Yaskawa INFORM job: A_ROOF_SIDE_0617_2_PAINT_56.JBI

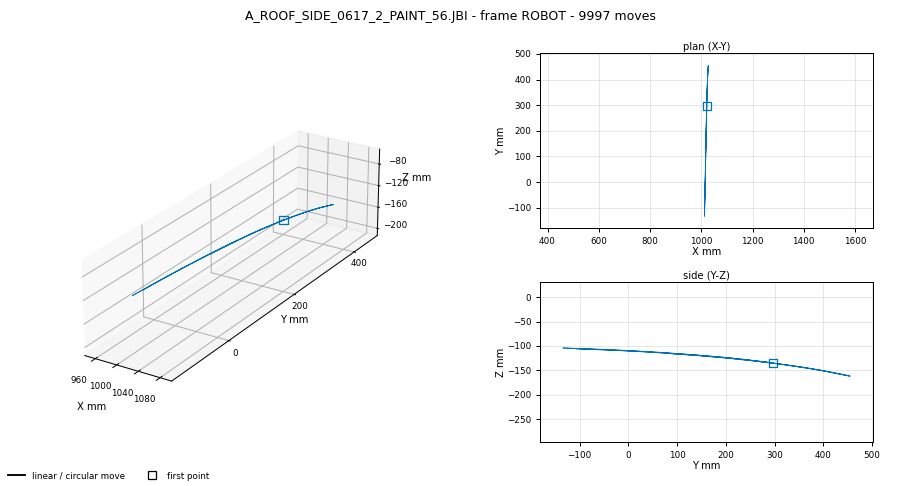
[picture p0: tool path of A_ROOF_SIDE_0617_2_PAINT_56.JBI in frame ROBOT, 9997 of 9997 moves have a stored position in this frame; points joined in program order, loops and branches not executed]
/JOB
//NAME A_ROOF_SIDE_0617_2_PAINT56
//POS
///NPOS 9997,0,0,0,0,0
///TOOL 1
///USER 0
///POSTYPE ROBOT
///RECTAN
///RCONF 1,0,0,0,0,0,0,0,0,0,0,0,0,0,0,0,0,0,0,0,0,0,0,0
C00000=1021.853,296.676,-134.515,170.306,49.131,159.506
C00001=1021.846,296.428,-134.484,170.301,49.134,159.506
C00002=1021.840,296.180,-134.452,170.296,49.136,159.506
C00003=1021.834,295.932,-134.419,170.291,49.139,159.506
C00004=1021.827,295.684,-134.388,170.287,49.142,159.506
C00005=1021.821,295.436,-134.355,170.281,49.145,159.506
C00006=1021.814,295.189,-134.324,170.276,49.148,159.506
C00007=1021.808,294.940,-134.292,170.271,49.151,159.506
C00008=1021.802,294.693,-134.259,170.266,49.153,159.505
C00009=1021.795,294.445,-134.227,170.261,49.156,159.505
C00010=1021.789,294.197,-134.195,170.256,49.159,159.505
C00011=1021.782,293.949,-134.163,170.251,49.162,159.505
C00012=1021.776,293.701,-134.131,170.246,49.165,159.505
C00013=1021.770,293.476,-134.103,170.242,49.168,159.505
C00014=1021.765,293.252,-134.073,170.237,49.170,159.505
C00015=1021.758,293.027,-134.045,170.233,49.173,159.505
C00016=1021.753,292.802,-134.016,170.227,49.176,159.505
C00017=1021.747,292.576,-133.987,170.223,49.179,159.505
C00018=1021.741,292.351,-133.959,170.219,49.182,159.505
C00019=1021.735,292.126,-133.931,170.214,49.184,159.504
C00020=1021.729,291.902,-133.901,170.210,49.187,159.504
C00021=1021.722,291.654,-133.870,170.204,49.190,159.504
C00022=1021.715,291.406,-133.838,170.200,49.193,159.504
C00023=1021.709,291.158,-133.807,170.195,49.196,159.504
C00024=1021.703,290.909,-133.776,170.189,49.199,159.504
C00025=1021.697,290.662,-133.745,170.185,49.202,159.504
C00026=1021.690,290.414,-133.713,170.180,49.205,159.504
C00027=1021.683,290.166,-133.682,170.174,49.209,159.504
C00028=1021.677,289.919,-133.650,170.170,49.211,159.504
C00029=1021.670,289.671,-133.619,170.165,49.215,159.504
C00030=1021.663,289.423,-133.588,170.161,49.218,159.504
C00031=1021.657,289.175,-133.556,170.155,49.221,159.504
C00032=1021.651,288.927,-133.525,170.150,49.225,159.504
C00033=1021.645,288.679,-133.494,170.146,49.227,159.504
C00034=1021.638,288.431,-133.462,170.140,49.231,159.504
C00035=1021.631,288.183,-133.431,170.135,49.234,159.504
C00036=1021.625,287.935,-133.400,170.131,49.237,159.504
C00037=1021.619,287.687,-133.369,170.126,49.241,159.504
C00038=1021.612,287.439,-133.338,170.122,49.243,159.504
C00039=1021.605,287.192,-133.306,170.116,49.247,159.504
C00040=1021.599,286.943,-133.275,170.111,49.250,159.504
C00041=1021.593,286.696,-133.244,170.107,49.253,159.504
C00042=1021.586,286.448,-133.213,170.102,49.257,159.504
C00043=1021.580,286.199,-133.182,170.096,49.260,159.504
C00044=1021.573,285.952,-133.151,170.092,49.263,159.504
C00045=1021.567,285.704,-133.120,170.087,49.267,159.504
C00046=1021.560,285.456,-133.089,170.083,49.269,159.504
C00047=1021.554,285.208,-133.058,170.078,49.273,159.504
C00048=1021.548,284.960,-133.027,170.072,49.277,159.504
C00049=1021.541,284.711,-132.997,170.068,49.279,159.504
C00050=1021.535,284.464,-132.965,170.063,49.283,159.504
C00051=1021.529,284.216,-132.935,170.058,49.286,159.504
C00052=1021.521,283.968,-132.904,170.054,49.290,159.504
C00053=1021.515,283.720,-132.873,170.048,49.293,159.504
C00054=1021.508,283.472,-132.842,170.043,49.297,159.504
C00055=1021.502,283.224,-132.811,170.039,49.300,159.504
C00056=1021.496,282.975,-132.781,170.034,49.304,159.504
C00057=1021.489,282.729,-132.750,170.029,49.307,159.504
C00058=1021.483,282.480,-132.720,170.025,49.311,159.504
C00059=1021.476,282.231,-132.689,170.020,49.314,159.504
C00060=1021.470,281.984,-132.658,170.016,49.317,159.504
C00061=1021.464,281.736,-132.627,170.010,49.321,159.504
C00062=1021.457,281.488,-132.597,170.005,49.324,159.504
C00063=1021.451,281.240,-132.567,170.001,49.327,159.504
C00064=1021.444,280.992,-132.535,169.996,49.331,159.504
C00065=1021.438,280.744,-132.505,169.991,49.335,159.504
C00066=1021.431,280.496,-132.475,169.987,49.338,159.504
C00067=1021.425,280.247,-132.444,169.982,49.342,159.504
C00068=1021.419,279.999,-132.414,169.978,49.345,159.504
C00069=1021.412,279.752,-132.382,169.972,49.349,159.504
C00070=1021.406,279.504,-132.352,169.967,49.352,159.504
C00071=1021.399,279.255,-132.322,169.963,49.356,159.505
C00072=1021.393,279.008,-132.291,169.958,49.359,159.505
C00073=1021.388,278.789,-132.264,169.954,49.363,159.505
C00074=1021.382,278.570,-132.238,169.950,49.366,159.505
C00075=1021.377,278.351,-132.210,169.946,49.369,159.505
C00076=1021.371,278.132,-132.183,169.942,49.372,159.505
C00077=1021.365,277.913,-132.157,169.937,49.375,159.505
C00078=1021.360,277.695,-132.130,169.933,49.379,159.505
C00079=1021.354,277.475,-132.103,169.930,49.381,159.505
C00080=1021.349,277.257,-132.076,169.926,49.384,159.505
C00081=1021.343,277.009,-132.046,169.921,49.388,159.505
C00082=1021.336,276.760,-132.015,169.916,49.392,159.505
C00083=1021.330,276.513,-131.985,169.912,49.395,159.505
C00084=1021.324,276.264,-131.954,169.907,49.399,159.506
C00085=1021.317,276.017,-131.925,169.902,49.403,159.506
C00086=1021.311,275.769,-131.894,169.898,49.407,159.506
C00087=1021.304,275.520,-131.865,169.893,49.411,159.506
C00088=1021.298,275.272,-131.835,169.889,49.414,159.506
C00089=1021.291,275.024,-131.804,169.884,49.417,159.506
C00090=1021.285,274.776,-131.774,169.879,49.421,159.506
C00091=1021.278,274.528,-131.744,169.875,49.425,159.506
C00092=1021.273,274.280,-131.714,169.870,49.429,159.506
C00093=1021.266,274.032,-131.685,169.865,49.433,159.506
C00094=1021.260,273.784,-131.654,169.861,49.436,159.507
C00095=1021.253,273.536,-131.624,169.856,49.440,159.507
C00096=1021.247,273.287,-131.594,169.852,49.444,159.507
C00097=1021.241,273.039,-131.564,169.847,49.447,159.507
C00098=1021.235,272.792,-131.534,169.842,49.451,159.507
C00099=1021.228,272.543,-131.503,169.838,49.455,159.507
C00100=1021.222,272.295,-131.474,169.833,49.459,159.507
C00101=1021.216,272.047,-131.445,169.828,49.463,159.508
C00102=1021.209,271.798,-131.415,169.824,49.467,159.508
C00103=1021.203,271.551,-131.385,169.819,49.471,159.508
C00104=1021.197,271.303,-131.354,169.814,49.475,159.508
C00105=1021.190,271.054,-131.325,169.811,49.478,159.508
C00106=1021.184,270.806,-131.295,169.806,49.482,159.508
C00107=1021.178,270.558,-131.266,169.802,49.486,159.508
C00108=1021.171,270.310,-131.235,169.797,49.490,159.509
C00109=1021.166,270.061,-131.206,169.792,49.494,159.509
C00110=1021.159,269.814,-131.176,169.788,49.498,159.509
C00111=1021.153,269.565,-131.146,169.783,49.502,159.509
C00112=1021.146,269.317,-131.116,169.778,49.506,159.509
C00113=1021.140,269.069,-131.087,169.775,49.510,159.509
C00114=1021.134,268.821,-131.057,169.770,49.514,159.510
C00115=1021.128,268.573,-131.028,169.766,49.517,159.510
C00116=1021.121,268.324,-130.998,169.761,49.522,159.510
C00117=1021.115,268.077,-130.969,169.756,49.526,159.510
C00118=1021.109,267.828,-130.939,169.752,49.529,159.510
C00119=1021.103,267.581,-130.909,169.748,49.534,159.511
C00120=1021.096,267.332,-130.880,169.743,49.538,159.511
C00121=1021.090,267.084,-130.850,169.739,49.541,159.511
C00122=1021.084,266.835,-130.821,169.734,49.546,159.511
C00123=1021.077,266.588,-130.792,169.729,49.550,159.511
C00124=1021.071,266.340,-130.762,169.725,49.553,159.511
C00125=1021.065,266.091,-130.732,169.720,49.558,159.512
C00126=1021.058,265.843,-130.703,169.717,49.561,159.512
C00127=1021.052,265.595,-130.674,169.712,49.566,159.512
C00128=1021.046,265.347,-130.645,169.707,49.570,159.512
C00129=1021.040,265.099,-130.616,169.703,49.574,159.513
C00130=1021.033,264.850,-130.586,169.698,49.578,159.513
C00131=1021.027,264.602,-130.557,169.694,49.583,159.513
C00132=1021.021,264.353,-130.528,169.690,49.586,159.513
C00133=1021.015,264.137,-130.502,169.686,49.590,159.513
C00134=1021.010,263.921,-130.476,169.682,49.593,159.513
C00135=1021.004,263.705,-130.451,169.678,49.598,159.514
C00136=1020.999,263.488,-130.425,169.674,49.601,159.514
C00137=1020.993,263.271,-130.400,169.670,49.605,159.514
C00138=1020.988,263.055,-130.374,169.667,49.608,159.514
C00139=1020.982,262.838,-130.349,169.663,49.612,159.514
C00140=1020.976,262.622,-130.324,169.659,49.615,159.515
C00141=1020.971,262.373,-130.294,169.654,49.620,159.515
C00142=1020.965,262.125,-130.265,169.650,49.624,159.515
C00143=1020.958,261.877,-130.236,169.645,49.628,159.515
C00144=1020.952,261.629,-130.207,169.642,49.632,159.516
C00145=1020.946,261.381,-130.178,169.637,49.636,159.516
C00146=1020.940,261.133,-130.149,169.632,49.641,159.516
C00147=1020.933,260.885,-130.120,169.629,49.645,159.516
C00148=1020.927,260.636,-130.091,169.624,49.649,159.516
C00149=1020.917,260.232,-130.044,169.617,49.656,159.517
C00150=1020.907,259.829,-129.997,169.609,49.664,159.517
C00151=1020.897,259.426,-129.951,169.602,49.671,159.518
C00152=1020.886,259.023,-129.904,169.596,49.678,159.518
C00153=1020.880,258.774,-129.875,169.591,49.682,159.519
C00154=1020.873,258.526,-129.846,169.586,49.687,159.519
C00155=1020.866,258.278,-129.818,169.583,49.691,159.519
C00156=1020.860,258.029,-129.790,169.578,49.695,159.519
C00157=1020.854,257.781,-129.761,169.574,49.700,159.520
C00158=1020.847,257.533,-129.732,169.569,49.705,159.520
C00159=1020.841,257.285,-129.704,169.566,49.709,159.520
C00160=1020.835,257.036,-129.675,169.561,49.713,159.521
C00161=1020.828,256.788,-129.647,169.556,49.718,159.521
C00162=1020.822,256.540,-129.618,169.553,49.722,159.521
C00163=1020.816,256.291,-129.590,169.548,49.727,159.522
C00164=1020.810,256.043,-129.561,169.544,49.731,159.522
C00165=1020.803,255.795,-129.532,169.539,49.736,159.522
C00166=1020.797,255.546,-129.504,169.535,49.740,159.522
C00167=1020.791,255.298,-129.475,169.531,49.745,159.523
C00168=1020.784,255.050,-129.447,169.526,49.749,159.523
C00169=1020.778,254.802,-129.418,169.523,49.754,159.523
C00170=1020.772,254.553,-129.390,169.518,49.758,159.524
C00171=1020.765,254.304,-129.362,169.514,49.764,159.524
C00172=1020.760,254.057,-129.333,169.509,49.768,159.524
C00173=1020.754,253.808,-129.305,169.506,49.772,159.525
C00174=1020.747,253.560,-129.277,169.501,49.777,159.525
C00175=1020.741,253.312,-129.248,169.497,49.782,159.525
C00176=1020.734,253.064,-129.219,169.493,49.786,159.526
C00177=1020.728,252.815,-129.191,169.488,49.790,159.526
C00178=1020.722,252.566,-129.163,169.484,49.796,159.526
C00179=1020.716,252.318,-129.134,169.480,49.800,159.527
C00180=1020.709,252.070,-129.106,169.476,49.805,159.527
C00181=1020.703,251.822,-129.078,169.471,49.809,159.527
C00182=1020.697,251.574,-129.049,169.467,49.814,159.528
C00183=1020.691,251.325,-129.022,169.463,49.818,159.528
C00184=1020.685,251.076,-128.993,169.459,49.823,159.528
C00185=1020.678,250.828,-128.964,169.455,49.828,159.529
C00186=1020.672,250.581,-128.937,169.450,49.833,159.529
C00187=1020.666,250.332,-128.909,169.446,49.837,159.529
C00188=1020.660,250.084,-128.880,169.442,49.842,159.530
C00189=1020.653,249.835,-128.852,169.438,49.847,159.530
C00190=1020.647,249.587,-128.823,169.434,49.851,159.530
C00191=1020.642,249.338,-128.796,169.430,49.856,159.531
C00192=1020.635,249.091,-128.767,169.425,49.861,159.531
C00193=1020.628,248.811,-128.736,169.421,49.866,159.532
C00194=1020.621,248.531,-128.704,169.416,49.872,159.532
C00195=1020.615,248.251,-128.671,169.411,49.876,159.532
C00196=1020.608,247.972,-128.640,169.406,49.882,159.533
C00197=1020.602,247.723,-128.612,169.403,49.887,159.533
C00198=1020.596,247.475,-128.584,169.398,49.891,159.534
C00199=1020.590,247.227,-128.556,169.394,49.896,159.534
C00200=1020.583,246.979,-128.528,169.390,49.901,159.534
C00201=1020.577,246.730,-128.499,169.386,49.906,159.535
C00202=1020.571,246.481,-128.471,169.381,49.910,159.535
C00203=1020.565,246.233,-128.444,169.378,49.915,159.535
C00204=1020.559,245.985,-128.415,169.374,49.920,159.536
C00205=1020.553,245.736,-128.388,169.369,49.925,159.536
C00206=1020.547,245.488,-128.360,169.365,49.930,159.536
C00207=1020.542,245.239,-128.331,169.362,49.935,159.537
C00208=1020.535,244.991,-128.304,169.357,49.939,159.537
C00209=1020.529,244.743,-128.276,169.353,49.944,159.538
C00210=1020.524,244.494,-128.247,169.349,49.949,159.538
C00211=1020.517,244.246,-128.220,169.345,49.953,159.538
C00212=1020.512,243.998,-128.192,169.340,49.959,159.539
C00213=1020.506,243.749,-128.163,169.337,49.963,159.539
C00214=1020.499,243.501,-128.136,169.333,49.968,159.540
C00215=1020.494,243.252,-128.108,169.329,49.974,159.540
C00216=1020.487,243.005,-128.080,169.324,49.978,159.540
C00217=1020.482,242.756,-128.052,169.321,49.983,159.541
C00218=1020.475,242.508,-128.024,169.316,49.988,159.541
C00219=1020.469,242.259,-127.997,169.312,49.993,159.542
C00220=1020.463,242.010,-127.969,169.308,49.998,159.542
C00221=1020.457,241.763,-127.942,169.304,50.003,159.543
C00222=1020.450,241.514,-127.914,169.300,50.008,159.543
C00223=1020.444,241.265,-127.886,169.296,50.013,159.543
C00224=1020.439,241.017,-127.859,169.292,50.018,159.544
C00225=1020.432,240.769,-127.831,169.288,50.023,159.544
C00226=1020.427,240.521,-127.803,169.284,50.028,159.545
C00227=1020.420,240.272,-127.776,169.280,50.033,159.545
C00228=1020.414,240.023,-127.748,169.276,50.039,159.546
C00229=1020.408,239.775,-127.721,169.271,50.043,159.546
C00230=1020.402,239.527,-127.693,169.268,50.048,159.546
C00231=1020.397,239.278,-127.666,169.264,50.054,159.547
C00232=1020.390,239.030,-127.638,169.259,50.059,159.547
C00233=1020.384,238.782,-127.611,169.255,50.064,159.548
C00234=1020.377,238.533,-127.584,169.252,50.069,159.548
C00235=1020.371,238.285,-127.556,169.248,50.074,159.549
C00236=1020.365,238.036,-127.529,169.243,50.079,159.549
C00237=1020.359,237.788,-127.502,169.239,50.084,159.550
C00238=1020.352,237.539,-127.475,169.235,50.090,159.550
C00239=1020.346,237.291,-127.448,169.231,50.095,159.551
C00240=1020.341,237.042,-127.420,169.228,50.100,159.551
C00241=1020.335,236.794,-127.393,169.223,50.105,159.552
C00242=1020.328,236.545,-127.366,169.219,50.110,159.552
C00243=1020.323,236.297,-127.339,169.215,50.116,159.552
C00244=1020.316,236.048,-127.311,169.211,50.121,159.553
C00245=1020.310,235.800,-127.284,169.207,50.126,159.553
C00246=1020.303,235.552,-127.257,169.204,50.131,159.554
C00247=1020.298,235.303,-127.230,169.199,50.137,159.554
C00248=1020.291,235.054,-127.203,169.195,50.142,159.555
C00249=1020.286,234.834,-127.179,169.192,50.147,159.555
C00250=1020.281,234.613,-127.155,169.188,50.151,159.556
C00251=1020.275,234.393,-127.130,169.184,50.157,159.556
C00252=1020.270,234.172,-127.107,169.181,50.161,159.557
C00253=1020.264,233.952,-127.082,169.178,50.166,159.557
C00254=1020.258,233.731,-127.059,169.174,50.171,159.558
C00255=1020.253,233.511,-127.035,169.171,50.175,159.558
C00256=1020.248,233.290,-127.011,169.167,50.181,159.559
C00257=1020.241,233.041,-126.984,169.163,50.186,159.559
C00258=1020.235,232.793,-126.957,169.159,50.191,159.560
C00259=1020.229,232.545,-126.930,169.155,50.196,159.560
C00260=1020.223,232.296,-126.903,169.151,50.201,159.560
C00261=1020.217,232.048,-126.876,169.147,50.207,159.561
C00262=1020.211,231.799,-126.849,169.143,50.213,159.562
C00263=1020.205,231.551,-126.822,169.139,50.218,159.562
C00264=1020.199,231.303,-126.795,169.136,50.223,159.563
C00265=1020.193,231.053,-126.768,169.131,50.228,159.563
C00266=1020.187,230.805,-126.742,169.128,50.234,159.564
C00267=1020.182,230.557,-126.714,169.124,50.240,159.564
C00268=1020.175,230.308,-126.687,169.119,50.245,159.565
C00269=1020.169,230.060,-126.661,169.115,50.250,159.565
C00270=1020.163,229.812,-126.634,169.111,50.256,159.566
C00271=1020.157,229.563,-126.607,169.108,50.261,159.566
C00272=1020.151,229.314,-126.580,169.104,50.267,159.567
C00273=1020.145,229.066,-126.554,169.100,50.273,159.567
C00274=1020.139,228.817,-126.527,169.096,50.278,159.568
C00275=1020.133,228.568,-126.500,169.092,50.283,159.568
C00276=1020.126,228.320,-126.474,169.088,50.289,159.569
C00277=1020.120,228.071,-126.447,169.084,50.295,159.569
C00278=1020.114,227.823,-126.420,169.080,50.301,159.570
C00279=1020.108,227.575,-126.394,169.076,50.306,159.571
C00280=1020.103,227.326,-126.367,169.073,50.311,159.571
C00281=1020.096,227.077,-126.340,169.069,50.317,159.572
C00282=1020.090,226.829,-126.313,169.065,50.322,159.572
C00283=1020.084,226.581,-126.287,169.061,50.328,159.573
C00284=1020.078,226.332,-126.261,169.057,50.334,159.573
C00285=1020.072,226.083,-126.234,169.053,50.340,159.574
C00286=1020.065,225.835,-126.208,169.049,50.345,159.575
C00287=1020.060,225.587,-126.181,169.045,50.351,159.575
C00288=1020.052,225.338,-126.154,169.042,50.357,159.576
C00289=1020.047,225.089,-126.129,169.037,50.363,159.576
C00290=1020.041,224.841,-126.102,169.034,50.369,159.577
C00291=1020.035,224.593,-126.076,169.030,50.375,159.578
C00292=1020.028,224.344,-126.049,169.026,50.380,159.578
C00293=1020.022,224.095,-126.023,169.022,50.386,159.579
C00294=1020.016,223.847,-125.997,169.018,50.391,159.579
C00295=1020.011,223.598,-125.970,169.014,50.397,159.580
C00296=1020.003,223.350,-125.944,169.010,50.403,159.581
C00297=1019.998,223.101,-125.918,169.006,50.409,159.581
C00298=1019.991,222.853,-125.892,169.003,50.414,159.582
C00299=1019.986,222.604,-125.865,169.000,50.420,159.582
C00300=1019.980,222.356,-125.838,168.996,50.426,159.583
C00301=1019.974,222.107,-125.813,168.992,50.432,159.584
C00302=1019.967,221.858,-125.786,168.988,50.438,159.584
C00303=1019.962,221.610,-125.759,168.984,50.444,159.585
C00304=1019.955,221.361,-125.734,168.980,50.449,159.585
C00305=1019.950,221.113,-125.708,168.976,50.455,159.586
C00306=1019.943,220.865,-125.681,168.972,50.461,159.587
C00307=1019.938,220.616,-125.656,168.969,50.467,159.587
C00308=1019.931,220.367,-125.628,168.965,50.473,159.588
C00309=1019.926,220.142,-125.606,168.961,50.479,159.588
C00310=1019.920,219.918,-125.582,168.958,50.484,159.589
C00311=1019.914,219.693,-125.558,168.954,50.489,159.589
C00312=1019.909,219.468,-125.535,168.950,50.494,159.590
C00313=1019.903,219.244,-125.511,168.948,50.500,159.591
C00314=1019.898,219.020,-125.487,168.943,50.505,159.591
C00315=1019.893,218.795,-125.464,168.940,50.510,159.592
C00316=1019.887,218.570,-125.440,168.938,50.516,159.592
C00317=1019.882,218.321,-125.414,168.933,50.521,159.593
C00318=1019.875,218.073,-125.388,168.930,50.527,159.594
C00319=1019.869,217.824,-125.363,168.926,50.533,159.594
C00320=1019.863,217.576,-125.336,168.921,50.540,159.595
C00321=1019.857,217.327,-125.311,168.917,50.546,159.595
C00322=1019.850,217.078,-125.285,168.914,50.552,159.596
C00323=1019.845,216.830,-125.258,168.910,50.558,159.597
C00324=1019.838,216.581,-125.233,168.907,50.565,159.598
C00325=1019.832,216.332,-125.208,168.903,50.571,159.598
C00326=1019.827,216.084,-125.181,168.899,50.577,159.599
C00327=1019.820,215.835,-125.156,168.895,50.583,159.600
C00328=1019.814,215.587,-125.130,168.892,50.589,159.600
C00329=1019.808,215.338,-125.104,168.888,50.595,159.601
C00330=1019.802,215.090,-125.078,168.884,50.601,159.602
C00331=1019.796,214.841,-125.053,168.880,50.607,159.602
C00332=1019.789,214.593,-125.027,168.877,50.613,159.603
C00333=1019.784,214.344,-125.001,168.873,50.619,159.604
C00334=1019.778,214.095,-124.976,168.869,50.625,159.604
C00335=1019.772,213.847,-124.950,168.866,50.632,159.605
C00336=1019.766,213.598,-124.924,168.861,50.638,159.606
C00337=1019.760,213.349,-124.898,168.857,50.644,159.606
C00338=1019.753,213.101,-124.873,168.853,50.650,159.607
C00339=1019.748,212.852,-124.847,168.850,50.656,159.608
C00340=1019.742,212.603,-124.822,168.846,50.662,159.608
C00341=1019.735,212.355,-124.796,168.843,50.669,159.609
C00342=1019.729,212.106,-124.770,168.839,50.675,159.610
C00343=1019.723,211.857,-124.744,168.835,50.681,159.610
C00344=1019.717,211.609,-124.719,168.831,50.687,159.611
C00345=1019.711,211.360,-124.694,168.828,50.694,159.612
C00346=1019.705,211.112,-124.667,168.824,50.700,159.613
C00347=1019.699,210.863,-124.642,168.821,50.706,159.613
C00348=1019.693,210.614,-124.616,168.816,50.713,159.614
C00349=1019.687,210.366,-124.591,168.813,50.719,159.615
C00350=1019.681,210.117,-124.565,168.809,50.726,159.615
C00351=1019.675,209.868,-124.540,168.805,50.732,159.616
C00352=1019.669,209.620,-124.515,168.802,50.738,159.617
C00353=1019.663,209.371,-124.490,168.798,50.744,159.617
C00354=1019.657,209.123,-124.464,168.794,50.751,159.618
C00355=1019.651,208.874,-124.439,168.791,50.757,159.619
C00356=1019.645,208.625,-124.414,168.786,50.764,159.620
C00357=1019.639,208.376,-124.388,168.783,50.770,159.620
C00358=1019.633,208.128,-124.362,168.779,50.777,159.621
C00359=1019.627,207.879,-124.337,168.775,50.783,159.622
C00360=1019.620,207.630,-124.312,168.772,50.789,159.623
C00361=1019.614,207.382,-124.286,168.768,50.795,159.623
C00362=1019.609,207.134,-124.261,168.764,50.803,159.624
C00363=1019.602,206.885,-124.236,168.760,50.809,159.625
C00364=1019.596,206.637,-124.211,168.757,50.815,159.626
C00365=1019.590,206.388,-124.185,168.753,50.821,159.626
C00366=1019.584,206.139,-124.160,168.750,50.828,159.627
C00367=1019.578,205.890,-124.135,168.747,50.835,159.628
C00368=1019.572,205.641,-124.110,168.742,50.841,159.628
C00369=1019.567,205.420,-124.087,168.739,50.847,159.629
C00370=1019.561,205.197,-124.065,168.736,50.853,159.630
C00371=1019.556,204.975,-124.043,168.733,50.859,159.631
C00372=1019.550,204.753,-124.021,168.729,50.865,159.631
C00373=1019.544,204.531,-123.998,168.726,50.871,159.632
C00374=1019.540,204.309,-123.975,168.723,50.877,159.633
C00375=1019.534,204.086,-123.953,168.719,50.883,159.633
C00376=1019.528,203.864,-123.931,168.716,50.889,159.634
C00377=1019.506,202.827,-123.833,168.258,50.794,159.534
C00378=1019.501,202.577,-123.810,168.254,50.801,159.535
C00379=1019.497,202.329,-123.786,168.250,50.809,159.535
C00380=1019.491,202.081,-123.763,168.245,50.817,159.536
C00381=1019.486,201.831,-123.739,168.241,50.824,159.537
C00382=1019.481,201.582,-123.716,168.237,50.832,159.538
C00383=1019.476,201.333,-123.692,168.231,50.839,159.538
C00384=1019.471,201.085,-123.670,168.227,50.847,159.539
C00385=1019.466,200.836,-123.645,168.223,50.854,159.540
C00386=1019.461,200.587,-123.622,168.219,50.862,159.541
C00387=1019.455,200.338,-123.599,168.214,50.869,159.542
C00388=1019.450,200.090,-123.576,168.209,50.877,159.542
C00389=1019.445,199.840,-123.552,168.205,50.884,159.543
C00390=1019.440,199.591,-123.529,168.201,50.892,159.544
C00391=1019.435,199.342,-123.506,168.197,50.899,159.545
C00392=1019.430,199.094,-123.483,168.192,50.907,159.545
C00393=1019.425,198.845,-123.460,168.188,50.915,159.546
C00394=1019.419,198.596,-123.437,168.183,50.922,159.547
C00395=1019.413,198.347,-123.414,168.178,50.931,159.548
C00396=1019.409,198.099,-123.390,168.174,50.938,159.549
C00397=1019.403,197.850,-123.368,168.170,50.946,159.550
C00398=1019.398,197.600,-123.345,168.166,50.953,159.550
C00399=1019.393,197.351,-123.322,168.161,50.962,159.551
C00400=1019.387,197.103,-123.299,168.157,50.970,159.552
C00401=1019.382,196.854,-123.276,168.153,50.977,159.553
C00402=1019.377,196.605,-123.253,168.148,50.985,159.554
C00403=1019.372,196.356,-123.230,168.144,50.993,159.555
C00404=1019.366,196.107,-123.208,168.140,51.001,159.556
C00405=1019.361,195.858,-123.184,168.135,51.008,159.556
C00406=1019.356,195.610,-123.162,168.130,51.016,159.557
C00407=1019.350,195.361,-123.139,168.126,51.024,159.558
C00408=1019.345,195.111,-123.115,168.122,51.031,159.559
C00409=1019.340,194.863,-123.093,168.118,51.039,159.560
C00410=1019.335,194.614,-123.070,168.114,51.047,159.560
C00411=1019.330,194.364,-123.047,168.109,51.055,159.561
C00412=1019.325,194.116,-123.025,168.105,51.062,159.562
C00413=1019.319,193.867,-123.002,168.101,51.070,159.563
C00414=1019.315,193.618,-122.979,168.097,51.078,159.564
C00415=1019.309,193.369,-122.956,168.093,51.085,159.565
C00416=1019.304,193.120,-122.934,168.088,51.093,159.565
C00417=1019.299,192.871,-122.911,168.084,51.101,159.566
C00418=1019.294,192.622,-122.888,168.080,51.109,159.567
C00419=1019.289,192.374,-122.866,168.075,51.116,159.568
C00420=1019.284,192.124,-122.842,168.071,51.124,159.569
C00421=1019.279,191.876,-122.820,168.066,51.132,159.570
C00422=1019.273,191.627,-122.797,168.062,51.140,159.570
C00423=1019.268,191.378,-122.774,168.058,51.147,159.571
C00424=1019.263,191.129,-122.752,168.054,51.155,159.572
C00425=1019.258,190.880,-122.729,168.050,51.163,159.573
C00426=1019.254,190.631,-122.707,168.046,51.170,159.574
C00427=1019.248,190.382,-122.684,168.042,51.178,159.575
C00428=1019.243,190.134,-122.661,168.037,51.186,159.575
C00429=1019.237,189.884,-122.639,168.033,51.194,159.576
C00430=1019.233,189.636,-122.616,168.029,51.201,159.577
C00431=1019.227,189.386,-122.593,168.025,51.209,159.578
C00432=1019.222,189.138,-122.571,168.021,51.217,159.579
C00433=1019.218,188.888,-122.548,168.017,51.225,159.580
C00434=1019.212,188.640,-122.525,168.013,51.232,159.580
C00435=1019.207,188.390,-122.503,168.009,51.240,159.581
C00436=1019.203,188.142,-122.480,168.005,51.248,159.582
C00437=1019.198,187.893,-122.458,168.001,51.256,159.583
C00438=1019.192,187.612,-122.432,167.996,51.264,159.584
C00439=1019.186,187.331,-122.407,167.991,51.273,159.585
C00440=1019.180,187.050,-122.381,167.987,51.282,159.586
C00441=1019.175,186.769,-122.356,167.982,51.291,159.587
C00442=1019.170,186.520,-122.334,167.978,51.298,159.588
C00443=1019.165,186.271,-122.312,167.974,51.306,159.589
C00444=1019.159,186.022,-122.289,167.970,51.314,159.590
C00445=1019.155,185.773,-122.266,167.965,51.322,159.590
C00446=1019.150,185.525,-122.244,167.961,51.329,159.591
C00447=1019.145,185.275,-122.222,167.957,51.337,159.592
C00448=1019.141,185.026,-122.199,167.953,51.345,159.593
C00449=1019.135,184.778,-122.176,167.949,51.353,159.594
C00450=1019.130,184.528,-122.154,167.945,51.360,159.594
C00451=1019.126,184.279,-122.132,167.941,51.368,159.595
C00452=1019.121,184.031,-122.109,167.937,51.376,159.596
C00453=1019.115,183.781,-122.087,167.933,51.384,159.597
C00454=1019.110,183.533,-122.065,167.929,51.391,159.598
C00455=1019.106,183.284,-122.042,167.925,51.399,159.599
C00456=1019.101,183.035,-122.020,167.921,51.407,159.600
C00457=1019.096,182.786,-121.998,167.917,51.415,159.601
C00458=1019.091,182.536,-121.975,167.913,51.422,159.601
C00459=1019.086,182.288,-121.952,167.910,51.430,159.602
C00460=1019.081,182.039,-121.931,167.906,51.438,159.603
C00461=1019.076,181.789,-121.908,167.901,51.446,159.604
C00462=1019.071,181.541,-121.886,167.897,51.454,159.605
C00463=1019.065,181.292,-121.865,167.893,51.462,159.606
C00464=1019.060,181.043,-121.843,167.889,51.470,159.607
C00465=1019.055,180.794,-121.821,167.885,51.478,159.608
C00466=1019.050,180.545,-121.801,167.882,51.486,159.609
C00467=1019.044,180.295,-121.778,167.878,51.494,159.610
C00468=1019.040,180.046,-121.756,167.873,51.502,159.610
C00469=1019.034,179.798,-121.735,167.869,51.510,159.611
C00470=1019.029,179.548,-121.713,167.865,51.518,159.612
C00471=1019.024,179.299,-121.691,167.862,51.527,159.613
C00472=1019.018,179.051,-121.670,167.858,51.535,159.614
C00473=1019.013,178.801,-121.648,167.854,51.543,159.615
C00474=1019.008,178.552,-121.626,167.850,51.551,159.616
C00475=1019.003,178.303,-121.605,167.846,51.559,159.617
C00476=1018.997,178.054,-121.583,167.842,51.566,159.618
C00477=1018.993,177.805,-121.561,167.838,51.574,159.619
C00478=1018.987,177.557,-121.540,167.834,51.582,159.620
C00479=1018.982,177.308,-121.518,167.830,51.591,159.620
C00480=1018.976,177.058,-121.497,167.826,51.599,159.621
C00481=1018.971,176.809,-121.475,167.822,51.607,159.622
C00482=1018.967,176.560,-121.453,167.818,51.615,159.623
C00483=1018.961,176.312,-121.432,167.814,51.623,159.624
C00484=1018.956,176.062,-121.411,167.811,51.631,159.625
C00485=1018.951,175.813,-121.389,167.807,51.639,159.626
C00486=1018.946,175.564,-121.367,167.803,51.647,159.627
C00487=1018.941,175.316,-121.346,167.799,51.655,159.628
C00488=1018.936,175.066,-121.324,167.795,51.663,159.629
C00489=1018.930,174.817,-121.303,167.791,51.671,159.630
C00490=1018.925,174.568,-121.281,167.787,51.679,159.631
C00491=1018.920,174.319,-121.260,167.784,51.687,159.632
C00492=1018.915,174.070,-121.238,167.780,51.695,159.632
C00493=1018.910,173.821,-121.217,167.776,51.703,159.633
C00494=1018.905,173.572,-121.196,167.772,51.711,159.634
C00495=1018.900,173.323,-121.174,167.768,51.719,159.635
C00496=1018.895,173.074,-121.152,167.764,51.727,159.636
C00497=1018.890,172.825,-121.131,167.761,51.736,159.637
C00498=1018.885,172.576,-121.110,167.757,51.744,159.638
C00499=1018.880,172.327,-121.088,167.753,51.752,159.639
C00500=1018.875,172.078,-121.067,167.749,51.760,159.640
C00501=1018.870,171.829,-121.045,167.746,51.768,159.641
C00502=1018.865,171.611,-121.026,167.742,51.775,159.642
C00503=1018.861,171.392,-121.008,167.739,51.782,159.642
C00504=1018.856,171.174,-120.989,167.736,51.788,159.643
C00505=1018.852,170.956,-120.970,167.733,51.795,159.644
C00506=1018.847,170.737,-120.951,167.729,51.802,159.645
C00507=1018.843,170.519,-120.932,167.726,51.809,159.646
C00508=1018.838,170.301,-120.915,167.722,51.817,159.646
C00509=1018.834,170.083,-120.896,167.719,51.824,159.647
C00510=1018.829,169.833,-120.874,167.715,51.832,159.648
C00511=1018.824,169.584,-120.853,167.712,51.839,159.649
C00512=1018.819,169.335,-120.831,167.709,51.848,159.650
C00513=1018.814,169.086,-120.810,167.705,51.856,159.651
C00514=1018.809,168.838,-120.789,167.701,51.864,159.652
C00515=1018.804,168.588,-120.768,167.697,51.872,159.653
C00516=1018.799,168.339,-120.746,167.693,51.880,159.654
C00517=1018.794,168.090,-120.725,167.690,51.888,159.655
C00518=1018.789,167.841,-120.703,167.686,51.896,159.656
C00519=1018.784,167.592,-120.683,167.682,51.904,159.657
C00520=1018.779,167.343,-120.661,167.678,51.912,159.657
C00521=1018.775,167.094,-120.640,167.675,51.920,159.658
C00522=1018.769,166.845,-120.619,167.672,51.928,159.659
C00523=1018.765,166.596,-120.597,167.668,51.936,159.660
C00524=1018.760,166.347,-120.576,167.664,51.944,159.661
C00525=1018.755,166.098,-120.555,167.660,51.952,159.662
C00526=1018.750,165.849,-120.534,167.656,51.960,159.663
C00527=1018.745,165.600,-120.513,167.652,51.968,159.664
C00528=1018.740,165.351,-120.491,167.649,51.976,159.665
C00529=1018.735,165.101,-120.470,167.646,51.984,159.666
C00530=1018.728,164.759,-120.441,167.640,51.995,159.667
C00531=1018.722,164.416,-120.412,167.636,52.006,159.669
C00532=1018.715,164.074,-120.383,167.631,52.017,159.670
C00533=1018.708,163.730,-120.354,167.626,52.028,159.671
C00534=1018.703,163.481,-120.332,167.622,52.036,159.672
C00535=1018.698,163.232,-120.312,167.618,52.044,159.673
C00536=1018.694,162.983,-120.291,167.616,52.052,159.674
C00537=1018.689,162.734,-120.269,167.612,52.060,159.675
C00538=1018.684,162.485,-120.248,167.608,52.068,159.676
C00539=1018.679,162.235,-120.227,167.604,52.076,159.677
C00540=1018.674,161.987,-120.207,167.600,52.084,159.678
C00541=1018.670,161.738,-120.185,167.598,52.092,159.679
C00542=1018.665,161.488,-120.164,167.594,52.100,159.680
C00543=1018.660,161.239,-120.143,167.590,52.108,159.680
C00544=1018.655,160.990,-120.122,167.586,52.116,159.681
C00545=1018.650,160.741,-120.101,167.584,52.124,159.682
C00546=1018.645,160.492,-120.080,167.580,52.132,159.683
C00547=1018.641,160.243,-120.058,167.576,52.140,159.684
C00548=1018.636,159.994,-120.038,167.572,52.148,159.685
C00549=1018.631,159.745,-120.016,167.570,52.156,159.686
C00550=1018.626,159.496,-119.996,167.566,52.164,159.687
C00551=1018.621,159.247,-119.975,167.562,52.172,159.688
C00552=1018.617,158.997,-119.954,167.558,52.180,159.689
C00553=1018.612,158.748,-119.933,167.556,52.188,159.690
C00554=1018.607,158.500,-119.913,167.552,52.196,159.691
C00555=1018.602,158.250,-119.892,167.548,52.204,159.692
C00556=1018.597,158.001,-119.871,167.545,52.213,159.693
C00557=1018.592,157.752,-119.851,167.541,52.221,159.694
C00558=1018.587,157.503,-119.830,167.537,52.229,159.695
C00559=1018.581,157.254,-119.809,167.534,52.237,159.696
C00560=1018.576,157.005,-119.789,167.531,52.245,159.697
C00561=1018.572,156.756,-119.769,167.527,52.253,159.698
C00562=1018.566,156.507,-119.748,167.524,52.261,159.699
C00563=1018.562,156.258,-119.727,167.520,52.269,159.699
C00564=1018.557,156.009,-119.706,167.516,52.278,159.701
C00565=1018.552,155.759,-119.687,167.513,52.286,159.702
C00566=1018.546,155.478,-119.664,167.509,52.295,159.703
C00567=1018.540,155.197,-119.640,167.506,52.305,159.704
C00568=1018.534,154.914,-119.617,167.501,52.314,159.705
C00569=1018.529,154.633,-119.594,167.497,52.323,159.706
C00570=1018.524,154.383,-119.574,167.494,52.331,159.707
C00571=1018.519,154.134,-119.553,167.491,52.340,159.708
C00572=1018.514,153.886,-119.533,167.487,52.348,159.709
C00573=1018.509,153.637,-119.513,167.483,52.356,159.710
C00574=1018.504,153.387,-119.491,167.480,52.364,159.711
C00575=1018.499,153.138,-119.471,167.477,52.372,159.712
C00576=1018.494,152.888,-119.451,167.474,52.381,159.713
C00577=1018.489,152.640,-119.431,167.470,52.389,159.714
C00578=1018.484,152.391,-119.410,167.466,52.397,159.715
C00579=1018.479,152.141,-119.390,167.463,52.406,159.716
C00580=1018.474,151.892,-119.370,167.460,52.413,159.717
C00581=1018.469,151.643,-119.350,167.456,52.421,159.718
C00582=1018.464,151.394,-119.330,167.453,52.430,159.719
C00583=1018.459,151.145,-119.309,167.449,52.438,159.720
C00584=1018.454,150.896,-119.289,167.446,52.446,159.721
C00585=1018.449,150.646,-119.269,167.443,52.454,159.722
C00586=1018.444,150.397,-119.249,167.440,52.463,159.723
C00587=1018.439,150.148,-119.228,167.436,52.471,159.724
C00588=1018.435,149.899,-119.209,167.432,52.479,159.725
C00589=1018.429,149.650,-119.188,167.429,52.488,159.726
C00590=1018.423,149.401,-119.168,167.426,52.496,159.727
C00591=1018.419,149.152,-119.149,167.423,52.504,159.728
C00592=1018.414,148.903,-119.128,167.419,52.512,159.729
C00593=1018.409,148.653,-119.108,167.416,52.521,159.730
C00594=1018.404,148.405,-119.088,167.413,52.529,159.731
C00595=1018.399,148.156,-119.068,167.409,52.537,159.732
C00596=1018.394,147.906,-119.048,167.406,52.545,159.733
C00597=1018.389,147.658,-119.028,167.402,52.554,159.734
C00598=1018.384,147.408,-119.008,167.399,52.562,159.735
C00599=1018.379,147.159,-118.987,167.396,52.570,159.736
C00600=1018.375,146.910,-118.968,167.393,52.578,159.737
C00601=1018.370,146.661,-118.947,167.389,52.587,159.738
C00602=1018.365,146.411,-118.927,167.385,52.595,159.739
C00603=1018.359,146.163,-118.908,167.383,52.602,159.740
C00604=1018.354,145.913,-118.888,167.379,52.611,159.741
C00605=1018.349,145.664,-118.867,167.376,52.619,159.742
C00606=1018.345,145.415,-118.848,167.372,52.628,159.743
C00607=1018.340,145.165,-118.828,167.370,52.636,159.744
C00608=1018.334,144.916,-118.808,167.366,52.644,159.745
C00609=1018.329,144.667,-118.789,167.363,52.653,159.746
C00610=1018.324,144.418,-118.768,167.359,52.661,159.747
C00611=1018.319,144.169,-118.749,167.355,52.669,159.748
C00612=1018.314,143.920,-118.729,167.353,52.678,159.749
C00613=1018.309,143.670,-118.709,167.350,52.686,159.750
C00614=1018.304,143.421,-118.689,167.346,52.694,159.751
C00615=1018.299,143.172,-118.670,167.343,52.703,159.752
C00616=1018.294,142.924,-118.650,167.339,52.711,159.753
C00617=1018.289,142.674,-118.630,167.337,52.720,159.754
C00618=1018.283,142.424,-118.611,167.333,52.728,159.755
C00619=1018.279,142.175,-118.591,167.329,52.736,159.756
C00620=1018.274,141.926,-118.571,167.326,52.745,159.757
C00621=1018.269,141.677,-118.552,167.324,52.753,159.758
C00622=1018.264,141.428,-118.532,167.320,52.761,159.759
C00623=1018.259,141.179,-118.513,167.317,52.770,159.760
C00624=1018.253,140.930,-118.493,167.313,52.778,159.761
C00625=1018.249,140.680,-118.473,167.310,52.786,159.762
C00626=1018.244,140.431,-118.453,167.307,52.795,159.763
C00627=1018.238,140.182,-118.434,167.304,52.803,159.764
C00628=1018.234,139.933,-118.414,167.301,52.811,159.765
C00629=1018.229,139.683,-118.394,167.298,52.819,159.766
C00630=1018.223,139.402,-118.372,167.294,52.829,159.767
C00631=1018.218,139.120,-118.350,167.291,52.838,159.769
C00632=1018.212,138.838,-118.328,167.287,52.848,159.770
C00633=1018.207,138.556,-118.306,167.282,52.857,159.771
C00634=1018.202,138.307,-118.286,167.280,52.865,159.772
C00635=1018.197,138.058,-118.267,167.276,52.873,159.773
C00636=1018.192,137.809,-118.247,167.273,52.882,159.774
C00637=1018.186,137.559,-118.228,167.271,52.890,159.775
C00638=1018.182,137.311,-118.208,167.267,52.898,159.776
C00639=1018.176,137.062,-118.189,167.264,52.907,159.777
C00640=1018.172,136.813,-118.169,167.260,52.915,159.778
C00641=1018.166,136.563,-118.150,167.258,52.923,159.779
C00642=1018.162,136.314,-118.130,167.254,52.932,159.780
C00643=1018.156,136.065,-118.111,167.251,52.940,159.781
C00644=1018.152,135.816,-118.092,167.248,52.949,159.782
C00645=1018.146,135.566,-118.073,167.245,52.957,159.783
C00646=1018.142,135.317,-118.053,167.241,52.965,159.784
C00647=1018.136,135.068,-118.034,167.238,52.974,159.785
C00648=1018.132,134.819,-118.014,167.235,52.982,159.786
C00649=1018.126,134.569,-117.995,167.232,52.991,159.787
C00650=1018.122,134.320,-117.976,167.229,52.999,159.788
C00651=1018.116,134.071,-117.956,167.226,53.008,159.790
C00652=1018.111,133.822,-117.937,167.223,53.016,159.791
C00653=1018.106,133.573,-117.918,167.219,53.024,159.791
C00654=1018.101,133.323,-117.899,167.216,53.033,159.793
C00655=1018.097,133.074,-117.880,167.213,53.041,159.794
C00656=1018.091,132.824,-117.861,167.211,53.050,159.795
C00657=1018.086,132.576,-117.842,167.207,53.058,159.796
C00658=1018.081,132.326,-117.822,167.203,53.066,159.797
C00659=1018.076,132.077,-117.803,167.201,53.075,159.798
C00660=1018.072,131.828,-117.784,167.198,53.083,159.799
C00661=1018.066,131.579,-117.764,167.194,53.092,159.800
C00662=1018.062,131.330,-117.745,167.192,53.100,159.801
C00663=1018.056,131.080,-117.726,167.188,53.108,159.802
C00664=1018.051,130.831,-117.708,167.185,53.117,159.803
C00665=1018.047,130.582,-117.688,167.182,53.125,159.804
C00666=1018.041,130.332,-117.669,167.179,53.133,159.805
C00667=1018.037,130.083,-117.649,167.176,53.142,159.806
C00668=1018.031,129.834,-117.630,167.172,53.150,159.807
C00669=1018.026,129.585,-117.612,167.170,53.159,159.808
C00670=1018.021,129.336,-117.593,167.167,53.167,159.809
C00671=1018.016,129.086,-117.573,167.163,53.176,159.810
C00672=1018.011,128.837,-117.555,167.160,53.184,159.811
C00673=1018.006,128.587,-117.536,167.158,53.193,159.813
C00674=1018.001,128.339,-117.517,167.154,53.201,159.813
C00675=1017.996,128.089,-117.499,167.151,53.210,159.815
C00676=1017.990,127.840,-117.480,167.148,53.219,159.816
C00677=1017.985,127.591,-117.461,167.145,53.227,159.817
C00678=1017.980,127.342,-117.443,167.142,53.236,159.818
C00679=1017.975,127.092,-117.423,167.139,53.244,159.819
C00680=1017.970,126.843,-117.405,167.136,53.253,159.820
C00681=1017.965,126.594,-117.386,167.133,53.261,159.821
C00682=1017.959,126.344,-117.368,167.130,53.270,159.822
C00683=1017.954,126.096,-117.349,167.126,53.278,159.823
C00684=1017.950,125.846,-117.331,167.123,53.287,159.824
C00685=1017.944,125.597,-117.311,167.121,53.295,159.825
C00686=1017.939,125.348,-117.293,167.118,53.304,159.826
C00687=1017.934,125.099,-117.274,167.114,53.312,159.827
C00688=1017.929,124.849,-117.255,167.111,53.321,159.828
C00689=1017.924,124.600,-117.236,167.108,53.329,159.830
C00690=1017.919,124.351,-117.218,167.105,53.338,159.831
C00691=1017.914,124.101,-117.199,167.102,53.346,159.832
C00692=1017.909,123.852,-117.180,167.100,53.355,159.833
C00693=1017.904,123.603,-117.162,167.096,53.363,159.834
C00694=1017.898,123.321,-117.141,167.092,53.373,159.835
C00695=1017.892,123.039,-117.120,167.090,53.383,159.836
C00696=1017.887,122.757,-117.099,167.086,53.392,159.837
C00697=1017.881,122.475,-117.078,167.083,53.402,159.839
C00698=1017.876,122.227,-117.059,167.080,53.410,159.840
C00699=1017.870,121.977,-117.040,167.076,53.419,159.841
C00700=1017.865,121.728,-117.021,167.073,53.427,159.842
C00701=1017.861,121.479,-117.003,167.071,53.436,159.843
C00702=1017.856,121.229,-116.985,167.067,53.444,159.844
C00703=1017.850,120.980,-116.966,167.064,53.453,159.845
C00704=1017.845,120.730,-116.948,167.062,53.461,159.846
C00705=1017.840,120.482,-116.929,167.059,53.470,159.847
C00706=1017.835,120.232,-116.911,167.055,53.478,159.848
C00707=1017.830,119.983,-116.891,167.053,53.486,159.849
C00708=1017.826,119.733,-116.873,167.050,53.495,159.850
C00709=1017.821,119.484,-116.855,167.047,53.503,159.851
C00710=1017.816,119.235,-116.836,167.044,53.512,159.853
C00711=1017.811,118.986,-116.818,167.040,53.520,159.854
C00712=1017.805,118.736,-116.798,167.038,53.529,159.855
C00713=1017.801,118.487,-116.780,167.035,53.537,159.856
C00714=1017.796,118.238,-116.762,167.031,53.546,159.857
C00715=1017.791,117.989,-116.743,167.029,53.554,159.858
C00716=1017.786,117.740,-116.725,167.026,53.563,159.859
C00717=1017.781,117.490,-116.706,167.023,53.572,159.860
C00718=1017.775,117.241,-116.688,167.020,53.579,159.861
C00719=1017.771,116.991,-116.669,167.017,53.588,159.862
C00720=1017.766,116.742,-116.651,167.015,53.596,159.863
C00721=1017.761,116.493,-116.632,167.011,53.605,159.864
C00722=1017.756,116.244,-116.614,167.008,53.614,159.865
C00723=1017.751,115.995,-116.596,167.006,53.622,159.866
C00724=1017.746,115.745,-116.577,167.002,53.630,159.867
C00725=1017.741,115.496,-116.559,167.000,53.639,159.869
C00726=1017.736,115.247,-116.540,166.997,53.647,159.869
C00727=1017.731,114.998,-116.522,166.993,53.655,159.870
C00728=1017.726,114.748,-116.503,166.991,53.664,159.872
C00729=1017.721,114.499,-116.485,166.988,53.672,159.873
C00730=1017.716,114.250,-116.466,166.985,53.680,159.874
C00731=1017.711,114.001,-116.448,166.982,53.689,159.875
C00732=1017.707,113.751,-116.429,166.980,53.697,159.876
C00733=1017.702,113.501,-116.411,166.976,53.705,159.877
C00734=1017.697,113.253,-116.392,166.973,53.714,159.878
C00735=1017.692,113.003,-116.374,166.971,53.722,159.879
C00736=1017.687,112.754,-116.356,166.967,53.731,159.880
C00737=1017.683,112.505,-116.338,166.965,53.739,159.881
C00738=1017.678,112.255,-116.319,166.962,53.748,159.882
C00739=1017.673,112.006,-116.300,166.960,53.756,159.883
C00740=1017.667,111.757,-116.283,166.957,53.765,159.884
C00741=1017.662,111.508,-116.265,166.953,53.773,159.885
C00742=1017.657,111.258,-116.246,166.951,53.782,159.887
C00743=1017.652,111.009,-116.228,166.948,53.790,159.887
C00744=1017.647,110.760,-116.211,166.945,53.799,159.889
C00745=1017.642,110.510,-116.192,166.942,53.807,159.890
C00746=1017.637,110.261,-116.174,166.939,53.816,159.891
C00747=1017.632,110.012,-116.157,166.936,53.824,159.892
C00748=1017.627,109.763,-116.138,166.934,53.833,159.893
C00749=1017.622,109.513,-116.120,166.930,53.841,159.894
C00750=1017.617,109.264,-116.102,166.928,53.850,159.895
C00751=1017.612,109.015,-116.085,166.925,53.858,159.896
C00752=1017.607,108.765,-116.066,166.922,53.867,159.897
C00753=1017.602,108.516,-116.049,166.918,53.876,159.898
C00754=1017.597,108.267,-116.031,166.916,53.885,159.900
C00755=1017.591,108.018,-116.013,166.913,53.893,159.900
C00756=1017.587,107.768,-115.996,166.910,53.902,159.902
C00757=1017.581,107.518,-115.977,166.908,53.910,159.903
C00758=1017.575,107.237,-115.957,166.904,53.920,159.904
C00759=1017.570,106.955,-115.937,166.902,53.930,159.905
C00760=1017.564,106.673,-115.917,166.898,53.939,159.906
C00761=1017.558,106.392,-115.897,166.895,53.949,159.908
C00762=1017.553,106.142,-115.879,166.892,53.958,159.909
C00763=1017.549,105.892,-115.861,166.889,53.967,159.910
C00764=1017.543,105.643,-115.844,166.887,53.975,159.911
C00765=1017.538,105.394,-115.826,166.883,53.984,159.912
C00766=1017.533,105.145,-115.808,166.880,53.993,159.913
C00767=1017.528,104.896,-115.790,166.878,54.001,159.914
C00768=1017.523,104.646,-115.773,166.875,54.009,159.915
C00769=1017.518,104.397,-115.755,166.872,54.018,159.916
C00770=1017.513,104.148,-115.737,166.869,54.026,159.917
C00771=1017.508,103.898,-115.719,166.866,54.035,159.919
C00772=1017.502,103.649,-115.702,166.864,54.043,159.920
C00773=1017.498,103.399,-115.684,166.861,54.052,159.921
C00774=1017.493,103.150,-115.666,166.857,54.061,159.922
C00775=1017.488,102.901,-115.648,166.856,54.069,159.923
C00776=1017.483,102.652,-115.630,166.852,54.078,159.924
C00777=1017.477,102.403,-115.613,166.850,54.086,159.925
C00778=1017.473,102.153,-115.595,166.847,54.095,159.926
C00779=1017.467,101.904,-115.578,166.843,54.103,159.927
C00780=1017.462,101.654,-115.559,166.842,54.112,159.928
C00781=1017.457,101.405,-115.542,166.838,54.120,159.929
C00782=1017.452,101.155,-115.524,166.836,54.129,159.931
C00783=1017.447,100.906,-115.507,166.833,54.137,159.932
C00784=1017.442,100.657,-115.489,166.830,54.146,159.933
C00785=1017.438,100.407,-115.472,166.828,54.154,159.934
C00786=1017.433,100.158,-115.454,166.824,54.163,159.935
C00787=1017.428,99.909,-115.436,166.822,54.172,159.936
C00788=1017.422,99.660,-115.418,166.819,54.180,159.937
C00789=1017.418,99.410,-115.401,166.817,54.189,159.938
C00790=1017.412,99.161,-115.383,166.814,54.197,159.939
C00791=1017.408,98.911,-115.366,166.810,54.206,159.940
C00792=1017.402,98.662,-115.348,166.808,54.214,159.941
C00793=1017.397,98.413,-115.331,166.805,54.223,159.943
C00794=1017.392,98.163,-115.314,166.802,54.232,159.944
C00795=1017.387,97.914,-115.296,166.800,54.240,159.945
C00796=1017.382,97.664,-115.279,166.797,54.249,159.946
C00797=1017.377,97.416,-115.262,166.794,54.258,159.947
C00798=1017.372,97.166,-115.245,166.792,54.266,159.948
C00799=1017.367,96.917,-115.227,166.789,54.275,159.949
C00800=1017.362,96.667,-115.210,166.785,54.284,159.950
C00801=1017.356,96.418,-115.192,166.783,54.292,159.951
C00802=1017.351,96.169,-115.175,166.780,54.301,159.952
C00803=1017.346,95.919,-115.157,166.777,54.310,159.954
C00804=1017.341,95.670,-115.140,166.775,54.318,159.955
C00805=1017.336,95.421,-115.124,166.772,54.327,159.956
C00806=1017.331,95.172,-115.106,166.770,54.335,159.957
C00807=1017.326,94.922,-115.089,166.767,54.344,159.958
C00808=1017.321,94.673,-115.071,166.763,54.353,159.959
C00809=1017.316,94.423,-115.054,166.761,54.361,159.960
C00810=1017.310,94.174,-115.037,166.758,54.370,159.961
C00811=1017.305,93.925,-115.020,166.755,54.379,159.962
C00812=1017.301,93.676,-115.002,166.753,54.387,159.963
C00813=1017.295,93.426,-114.985,166.750,54.396,159.965
C00814=1017.290,93.176,-114.969,166.748,54.404,159.966
C00815=1017.285,92.927,-114.951,166.744,54.413,159.967
C00816=1017.280,92.677,-114.934,166.741,54.422,159.968
C00817=1017.275,92.429,-114.916,166.739,54.430,159.969
C00818=1017.270,92.179,-114.899,166.736,54.439,159.970
C00819=1017.265,91.930,-114.883,166.734,54.447,159.971
C00820=1017.260,91.680,-114.864,166.731,54.456,159.972
C00821=1017.255,91.431,-114.848,166.728,54.465,159.973
C00822=1017.249,91.149,-114.828,166.725,54.474,159.975
C00823=1017.243,90.868,-114.809,166.723,54.484,159.976
C00824=1017.238,90.586,-114.789,166.719,54.494,159.977
C00825=1017.233,90.305,-114.770,166.716,54.503,159.978
C00826=1017.227,90.055,-114.753,166.713,54.511,159.979
C00827=1017.222,89.806,-114.736,166.711,54.520,159.981
C00828=1017.217,89.556,-114.718,166.708,54.529,159.981
C00829=1017.212,89.307,-114.701,166.705,54.538,159.983
C00830=1017.208,89.058,-114.685,166.703,54.546,159.984
C00831=1017.202,88.808,-114.668,166.699,54.554,159.985
C00832=1017.197,88.559,-114.650,166.698,54.563,159.986
C00833=1017.192,88.309,-114.634,166.694,54.572,159.987
C00834=1017.187,88.060,-114.617,166.691,54.581,159.988
C00835=1017.182,87.811,-114.600,166.690,54.590,159.989
C00836=1017.177,87.561,-114.583,166.686,54.598,159.990
C00837=1017.171,87.311,-114.567,166.684,54.607,159.992
C00838=1017.167,87.062,-114.550,166.681,54.615,159.993
C00839=1017.162,86.813,-114.533,166.678,54.624,159.994
C00840=1017.156,86.564,-114.516,166.675,54.633,159.995
C00841=1017.150,86.314,-114.499,166.673,54.642,159.996
C00842=1017.145,86.065,-114.483,166.670,54.650,159.997
C00843=1017.140,85.816,-114.466,166.667,54.659,159.998
C00844=1017.135,85.566,-114.449,166.665,54.667,159.999
C00845=1017.130,85.316,-114.432,166.662,54.677,160.000
C00846=1017.125,85.067,-114.416,166.659,54.685,160.001
C00847=1017.120,84.818,-114.399,166.657,54.694,160.003
C00848=1017.115,84.568,-114.382,166.654,54.702,160.004
C00849=1017.110,84.319,-114.366,166.652,54.711,160.005
C00850=1017.105,84.069,-114.349,166.649,54.720,160.006
C00851=1017.100,83.820,-114.332,166.645,54.728,160.007
C00852=1017.095,83.571,-114.316,166.644,54.737,160.008
C00853=1017.089,83.322,-114.299,166.640,54.745,160.009
C00854=1017.084,83.072,-114.282,166.638,54.755,160.010
C00855=1017.079,82.823,-114.266,166.635,54.763,160.011
C00856=1017.074,82.573,-114.249,166.633,54.772,160.013
C00857=1017.069,82.324,-114.232,166.630,54.780,160.014
C00858=1017.064,82.075,-114.216,166.628,54.789,160.015
C00859=1017.059,81.825,-114.199,166.624,54.798,160.016
C00860=1017.054,81.575,-114.182,166.622,54.806,160.017
C00861=1017.049,81.326,-114.166,166.619,54.815,160.018
C00862=1017.044,81.077,-114.149,166.617,54.823,160.019
C00863=1017.039,80.827,-114.132,166.614,54.832,160.020
C00864=1017.033,80.578,-114.116,166.612,54.840,160.021
C00865=1017.028,80.329,-114.099,166.609,54.849,160.022
C00866=1017.023,80.079,-114.082,166.606,54.858,160.024
C00867=1017.018,79.830,-114.066,166.604,54.866,160.025
C00868=1017.013,79.580,-114.049,166.600,54.875,160.026
C00869=1017.009,79.331,-114.032,166.599,54.884,160.027
C00870=1017.003,79.082,-114.016,166.596,54.892,160.028
C00871=1016.998,78.832,-113.999,166.593,54.900,160.029
C00872=1016.994,78.583,-113.982,166.591,54.909,160.030
C00873=1016.988,78.334,-113.965,166.587,54.918,160.031
C00874=1016.983,78.085,-113.950,166.585,54.926,160.032
C00875=1016.978,77.835,-113.933,166.582,54.935,160.033
C00876=1016.973,77.586,-113.916,166.580,54.943,160.034
C00877=1016.968,77.337,-113.899,166.577,54.952,160.035
C00878=1016.963,77.086,-113.883,166.575,54.961,160.037
C00879=1016.958,76.837,-113.867,166.572,54.969,160.038
C00880=1016.953,76.588,-113.850,166.569,54.979,160.039
C00881=1016.947,76.338,-113.834,166.567,54.987,160.040
C00882=1016.943,76.089,-113.817,166.564,54.995,160.041
C00883=1016.938,75.839,-113.801,166.562,55.004,160.042
C00884=1016.932,75.591,-113.785,166.559,55.013,160.043
C00885=1016.927,75.341,-113.768,166.556,55.022,160.044
C00886=1016.922,75.059,-113.750,166.553,55.031,160.046
C00887=1016.916,74.778,-113.732,166.550,55.041,160.047
C00888=1016.910,74.495,-113.713,166.547,55.051,160.048
C00889=1016.904,74.215,-113.695,166.544,55.061,160.049
C00890=1016.899,73.965,-113.679,166.542,55.069,160.050
C00891=1016.894,73.716,-113.663,166.539,55.078,160.052
C00892=1016.889,73.466,-113.646,166.537,55.087,160.053
C00893=1016.884,73.216,-113.630,166.534,55.095,160.054
C00894=1016.878,72.967,-113.614,166.531,55.104,160.055
C00895=1016.873,72.718,-113.597,166.529,55.112,160.056
C00896=1016.868,72.469,-113.582,166.526,55.122,160.057
C00897=1016.863,72.219,-113.565,166.524,55.130,160.058
C00898=1016.858,71.970,-113.549,166.521,55.138,160.059
C00899=1016.853,71.720,-113.533,166.518,55.148,160.060
C00900=1016.848,71.471,-113.517,166.516,55.156,160.062
C00901=1016.842,71.222,-113.500,166.513,55.164,160.062
C00902=1016.838,70.972,-113.485,166.511,55.173,160.064
C00903=1016.833,70.722,-113.468,166.508,55.182,160.065
C00904=1016.828,70.473,-113.453,166.505,55.190,160.066
C00905=1016.822,70.223,-113.436,166.503,55.199,160.067
C00906=1016.817,69.974,-113.421,166.500,55.208,160.068
C00907=1016.812,69.725,-113.404,166.498,55.217,160.069
C00908=1016.807,69.476,-113.388,166.495,55.225,160.070
C00909=1016.802,69.226,-113.372,166.493,55.233,160.071
C00910=1016.797,68.977,-113.355,166.490,55.243,160.073
C00911=1016.792,68.727,-113.340,166.487,55.251,160.074
C00912=1016.787,68.478,-113.323,166.485,55.259,160.075
C00913=1016.782,68.228,-113.308,166.482,55.268,160.076
C00914=1016.777,67.979,-113.291,166.480,55.277,160.077
C00915=1016.772,67.730,-113.276,166.477,55.285,160.078
C00916=1016.766,67.480,-113.259,166.474,55.295,160.079
C00917=1016.761,67.231,-113.244,166.472,55.303,160.080
C00918=1016.755,66.981,-113.228,166.469,55.311,160.081
C00919=1016.751,66.732,-113.212,166.467,55.320,160.083
C00920=1016.746,66.482,-113.196,166.464,55.329,160.083
C00921=1016.741,66.233,-113.180,166.461,55.337,160.084
C00922=1016.735,65.983,-113.164,166.459,55.346,160.086
C00923=1016.731,65.734,-113.148,166.456,55.355,160.087
C00924=1016.726,65.485,-113.133,166.454,55.363,160.088
C00925=1016.720,65.235,-113.117,166.451,55.372,160.089
C00926=1016.715,64.986,-113.101,166.448,55.381,160.090
C00927=1016.710,64.736,-113.085,166.446,55.390,160.091
C00928=1016.704,64.487,-113.069,166.443,55.398,160.092
C00929=1016.700,64.237,-113.054,166.441,55.407,160.093
C00930=1016.694,63.987,-113.038,166.439,55.416,160.095
C00931=1016.690,63.739,-113.022,166.435,55.424,160.096
C00932=1016.684,63.489,-113.006,166.433,55.433,160.097
C00933=1016.679,63.239,-112.991,166.430,55.441,160.098
C00934=1016.674,62.990,-112.974,166.429,55.450,160.099
C00935=1016.669,62.740,-112.959,166.425,55.459,160.100
C00936=1016.664,62.491,-112.944,166.423,55.468,160.101
C00937=1016.658,62.241,-112.928,166.421,55.476,160.102
C00938=1016.653,61.992,-112.913,166.418,55.486,160.104
C00939=1016.647,61.742,-112.897,166.415,55.494,160.104
C00940=1016.642,61.493,-112.881,166.412,55.504,160.106
C00941=1016.637,61.244,-112.866,166.410,55.512,160.107
C00942=1016.632,60.994,-112.850,166.408,55.521,160.108
C00943=1016.627,60.744,-112.835,166.404,55.530,160.109
C00944=1016.622,60.495,-112.820,166.402,55.538,160.110
C00945=1016.616,60.245,-112.804,166.400,55.547,160.111
C00946=1016.611,59.996,-112.789,166.397,55.556,160.112
C00947=1016.606,59.747,-112.774,166.394,55.565,160.113
C00948=1016.600,59.497,-112.758,166.392,55.573,160.115
C00949=1016.595,59.248,-112.742,166.389,55.583,160.116
C00950=1016.590,58.966,-112.726,166.387,55.592,160.117
C00951=1016.584,58.684,-112.708,166.384,55.602,160.118
C00952=1016.578,58.403,-112.691,166.381,55.612,160.120
C00953=1016.572,58.122,-112.674,166.378,55.622,160.121
C00954=1016.566,57.872,-112.658,166.375,55.631,160.122
C00955=1016.562,57.622,-112.642,166.373,55.639,160.123
C00956=1016.557,57.373,-112.627,166.370,55.648,160.124
C00957=1016.551,57.123,-112.612,166.367,55.657,160.125
C00958=1016.546,56.874,-112.596,166.365,55.665,160.126
C00959=1016.541,56.625,-112.581,166.362,55.675,160.127
C00960=1016.535,56.375,-112.566,166.359,55.683,160.128
C00961=1016.530,56.125,-112.550,166.358,55.692,160.130
C00962=1016.525,55.876,-112.535,166.355,55.701,160.131
C00963=1016.520,55.627,-112.520,166.351,55.709,160.132
C00964=1016.514,55.377,-112.505,166.349,55.718,160.133
C00965=1016.509,55.128,-112.489,166.347,55.727,160.134
C00966=1016.504,54.878,-112.474,166.345,55.735,160.135
C00967=1016.499,54.628,-112.459,166.342,55.744,160.136
C00968=1016.494,54.379,-112.444,166.339,55.753,160.137
C00969=1016.489,54.130,-112.428,166.337,55.761,160.138
C00970=1016.484,53.881,-112.413,166.334,55.770,160.139
C00971=1016.478,53.631,-112.398,166.331,55.779,160.141
C00972=1016.473,53.381,-112.382,166.329,55.788,160.142
C00973=1016.468,53.132,-112.367,166.326,55.796,160.143
C00974=1016.463,52.883,-112.352,166.324,55.805,160.144
C00975=1016.457,52.633,-112.337,166.322,55.814,160.145
C00976=1016.452,52.384,-112.321,166.319,55.823,160.146
C00977=1016.447,52.134,-112.306,166.317,55.831,160.147
C00978=1016.443,51.885,-112.290,166.313,55.839,160.148
C00979=1016.438,51.635,-112.275,166.311,55.848,160.149
C00980=1016.432,51.385,-112.260,166.309,55.857,160.150
C00981=1016.427,51.136,-112.245,166.307,55.865,160.152
C00982=1016.422,50.886,-112.230,166.304,55.874,160.152
C00983=1016.417,50.637,-112.215,166.301,55.883,160.153
C00984=1016.412,50.388,-112.200,166.299,55.891,160.155
C00985=1016.407,50.138,-112.184,166.296,55.900,160.156
C00986=1016.402,49.889,-112.169,166.294,55.908,160.157
C00987=1016.397,49.639,-112.154,166.291,55.917,160.158
C00988=1016.391,49.390,-112.139,166.289,55.925,160.159
C00989=1016.387,49.140,-112.124,166.286,55.934,160.160
C00990=1016.381,48.890,-112.109,166.283,55.943,160.161
C00991=1016.376,48.641,-112.094,166.281,55.951,160.162
C00992=1016.371,48.392,-112.078,166.278,55.960,160.163
C00993=1016.366,48.142,-112.063,166.276,55.969,160.164
C00994=1016.361,47.893,-112.048,166.273,55.977,160.165
C00995=1016.356,47.644,-112.033,166.271,55.986,160.167
C00996=1016.351,47.393,-112.018,166.268,55.994,160.167
C00997=1016.345,47.144,-112.003,166.266,56.002,160.169
C00998=1016.340,46.895,-111.988,166.263,56.011,160.170
C00999=1016.335,46.645,-111.972,166.261,56.019,160.171
C01000=1016.330,46.396,-111.957,166.258,56.028,160.172
C01001=1016.326,46.146,-111.943,166.256,56.036,160.173
C01002=1016.321,45.897,-111.928,166.253,56.045,160.174
C01003=1016.315,45.647,-111.912,166.251,56.053,160.175
C01004=1016.310,45.398,-111.897,166.248,56.062,160.176
C01005=1016.305,45.149,-111.882,166.246,56.070,160.177
C01006=1016.300,44.899,-111.867,166.243,56.079,160.178
C01007=1016.295,44.649,-111.852,166.241,56.087,160.179
C01008=1016.290,44.400,-111.837,166.238,56.096,160.180
C01009=1016.285,44.151,-111.822,166.236,56.104,160.181
C01010=1016.280,43.901,-111.807,166.233,56.113,160.182
C01011=1016.276,43.651,-111.792,166.231,56.121,160.183
C01012=1016.271,43.402,-111.776,166.228,56.130,160.184
C01013=1016.265,43.152,-111.761,166.226,56.138,160.185
C01014=1016.259,42.871,-111.745,166.223,56.148,160.186
C01015=1016.254,42.589,-111.728,166.220,56.157,160.188
C01016=1016.248,42.307,-111.711,166.218,56.167,160.189
C01017=1016.243,42.026,-111.694,166.214,56.177,160.190
C01018=1016.238,41.776,-111.679,166.212,56.185,160.191
C01019=1016.232,41.527,-111.665,166.209,56.194,160.192
C01020=1016.227,41.277,-111.650,166.208,56.203,160.194
C01021=1016.222,41.028,-111.635,166.205,56.211,160.195
C01022=1016.217,40.779,-111.620,166.203,56.220,160.196
C01023=1016.212,40.529,-111.606,166.200,56.228,160.197
C01024=1016.207,40.279,-111.591,166.197,56.237,160.198
C01025=1016.202,40.030,-111.576,166.195,56.245,160.199
C01026=1016.196,39.781,-111.562,166.192,56.254,160.200
C01027=1016.192,39.531,-111.547,166.190,56.262,160.201
C01028=1016.187,39.281,-111.532,166.187,56.271,160.202
C01029=1016.182,39.032,-111.518,166.185,56.279,160.203
C01030=1016.176,38.783,-111.503,166.182,56.288,160.204
C01031=1016.171,38.533,-111.489,166.180,56.296,160.205
C01032=1016.166,38.283,-111.474,166.177,56.305,160.206
C01033=1016.161,38.034,-111.460,166.174,56.314,160.207
C01034=1016.156,37.785,-111.444,166.172,56.322,160.208
C01035=1016.151,37.535,-111.430,166.169,56.331,160.209
C01036=1016.146,37.285,-111.415,166.167,56.339,160.210
C01037=1016.140,37.036,-111.401,166.164,56.348,160.211
C01038=1016.135,36.785,-111.386,166.163,56.356,160.212
C01039=1016.130,36.536,-111.371,166.160,56.365,160.213
C01040=1016.125,36.286,-111.357,166.158,56.373,160.214
C01041=1016.120,36.037,-111.342,166.155,56.382,160.215
C01042=1016.114,35.788,-111.328,166.152,56.391,160.217
C01043=1016.109,35.538,-111.314,166.150,56.400,160.218
C01044=1016.104,35.288,-111.300,166.147,56.408,160.219
C01045=1016.099,35.039,-111.285,166.145,56.417,160.220
C01046=1016.094,34.790,-111.271,166.142,56.425,160.221
C01047=1016.089,34.540,-111.257,166.140,56.434,160.222
C01048=1016.083,34.291,-111.242,166.138,56.442,160.223
C01049=1016.079,34.041,-111.228,166.135,56.451,160.224
C01050=1016.073,33.792,-111.214,166.133,56.460,160.225
C01051=1016.068,33.542,-111.199,166.130,56.468,160.226
C01052=1016.063,33.293,-111.185,166.127,56.477,160.227
C01053=1016.058,33.043,-111.170,166.125,56.485,160.228
C01054=1016.052,32.793,-111.156,166.122,56.494,160.229
C01055=1016.048,32.543,-111.142,166.120,56.502,160.230
C01056=1016.042,32.294,-111.128,166.117,56.511,160.231
C01057=1016.037,32.045,-111.113,166.114,56.520,160.232
C01058=1016.032,31.795,-111.099,166.112,56.528,160.234
C01059=1016.027,31.545,-111.085,166.109,56.537,160.234
C01060=1016.022,31.296,-111.071,166.108,56.545,160.236
C01061=1016.016,31.046,-111.057,166.105,56.554,160.237
C01062=1016.012,30.797,-111.042,166.103,56.562,160.238
C01063=1016.006,30.548,-111.028,166.100,56.571,160.239
C01064=1016.001,30.298,-111.014,166.098,56.579,160.240
C01065=1015.996,30.048,-111.000,166.095,56.588,160.241
C01066=1015.991,29.799,-110.985,166.092,56.597,160.242
C01067=1015.986,29.549,-110.971,166.090,56.605,160.243
C01068=1015.981,29.300,-110.956,166.087,56.614,160.244
C01069=1015.975,29.050,-110.942,166.085,56.622,160.245
C01070=1015.970,28.800,-110.928,166.082,56.631,160.246
C01071=1015.966,28.551,-110.914,166.081,56.640,160.247
C01072=1015.961,28.301,-110.900,166.077,56.648,160.248
C01073=1015.955,28.052,-110.886,166.075,56.656,160.249
C01074=1015.951,27.802,-110.872,166.072,56.665,160.250
C01075=1015.945,27.552,-110.858,166.070,56.673,160.251
C01076=1015.939,27.304,-110.843,166.068,56.682,160.252
C01077=1015.935,27.054,-110.829,166.066,56.690,160.253
C01078=1015.929,26.772,-110.814,166.062,56.700,160.255
C01079=1015.923,26.490,-110.798,166.060,56.710,160.256
C01080=1015.917,26.209,-110.782,166.057,56.720,160.257
C01081=1015.912,25.927,-110.766,166.054,56.729,160.258
C01082=1015.907,25.678,-110.752,166.051,56.738,160.259
C01083=1015.901,25.428,-110.739,166.050,56.746,160.260
C01084=1015.896,25.179,-110.725,166.046,56.754,160.261
C01085=1015.891,24.929,-110.710,166.044,56.763,160.262
C01086=1015.886,24.680,-110.697,166.041,56.771,160.263
C01087=1015.881,24.430,-110.683,166.038,56.780,160.264
C01088=1015.875,24.181,-110.669,166.037,56.788,160.265
C01089=1015.870,23.931,-110.655,166.034,56.797,160.266
C01090=1015.865,23.681,-110.641,166.032,56.806,160.267
C01091=1015.860,23.432,-110.628,166.029,56.814,160.268
C01092=1015.855,23.182,-110.614,166.027,56.823,160.270
C01093=1015.849,22.933,-110.600,166.024,56.832,160.271
C01094=1015.845,22.683,-110.586,166.021,56.840,160.271
C01095=1015.839,22.433,-110.572,166.019,56.848,160.272
C01096=1015.834,22.184,-110.558,166.016,56.857,160.273
C01097=1015.829,21.935,-110.545,166.014,56.865,160.275
C01098=1015.823,21.685,-110.531,166.011,56.874,160.276
C01099=1015.819,21.435,-110.517,166.010,56.882,160.277
C01100=1015.814,21.186,-110.503,166.006,56.890,160.277
C01101=1015.808,20.936,-110.490,166.004,56.899,160.279
C01102=1015.803,20.687,-110.476,166.002,56.908,160.280
C01103=1015.798,20.437,-110.461,166.000,56.916,160.281
C01104=1015.793,20.188,-110.448,165.997,56.925,160.282
C01105=1015.788,19.938,-110.435,165.994,56.932,160.283
C01106=1015.783,19.688,-110.421,165.992,56.941,160.284
C01107=1015.777,19.439,-110.407,165.990,56.950,160.285
C01108=1015.773,19.189,-110.393,165.987,56.958,160.286
C01109=1015.768,18.940,-110.379,165.985,56.966,160.287
C01110=1015.762,18.690,-110.366,165.982,56.975,160.288
C01111=1015.758,18.441,-110.352,165.979,56.984,160.289
C01112=1015.752,18.191,-110.338,165.977,56.992,160.290
C01113=1015.747,17.941,-110.325,165.974,57.001,160.291
C01114=1015.741,17.691,-110.311,165.972,57.009,160.292
C01115=1015.737,17.443,-110.298,165.969,57.017,160.293
C01116=1015.731,17.192,-110.285,165.967,57.026,160.294
C01117=1015.726,16.943,-110.271,165.964,57.035,160.295
C01118=1015.721,16.694,-110.257,165.963,57.043,160.296
C01119=1015.716,16.444,-110.244,165.959,57.051,160.297
C01120=1015.710,16.194,-110.230,165.956,57.060,160.298
C01121=1015.706,15.945,-110.217,165.955,57.068,160.299
C01122=1015.701,15.695,-110.203,165.952,57.077,160.300
C01123=1015.696,15.445,-110.189,165.949,57.085,160.301
C01124=1015.691,15.196,-110.176,165.947,57.094,160.302
C01125=1015.686,14.946,-110.163,165.945,57.102,160.303
C01126=1015.680,14.697,-110.149,165.941,57.110,160.304
C01127=1015.676,14.447,-110.136,165.940,57.119,160.305
C01128=1015.670,14.197,-110.122,165.937,57.127,160.306
C01129=1015.665,13.948,-110.108,165.935,57.135,160.307
C01130=1015.660,13.698,-110.095,165.932,57.144,160.308
C01131=1015.655,13.449,-110.082,165.930,57.152,160.309
C01132=1015.649,13.199,-110.068,165.927,57.160,160.310
C01133=1015.645,12.950,-110.055,165.925,57.169,160.311
C01134=1015.639,12.700,-110.042,165.922,57.178,160.312
C01135=1015.634,12.450,-110.028,165.920,57.186,160.313
C01136=1015.629,12.201,-110.016,165.917,57.195,160.314
C01137=1015.623,11.951,-110.003,165.914,57.203,160.315
C01138=1015.619,11.702,-109.989,165.912,57.212,160.316
C01139=1015.613,11.452,-109.976,165.910,57.220,160.317
C01140=1015.607,11.202,-109.963,165.908,57.229,160.318
C01141=1015.603,10.953,-109.950,165.904,57.237,160.319
C01142=1015.595,10.603,-109.931,165.901,57.249,160.320
C01143=1015.588,10.253,-109.913,165.897,57.261,160.321
C01144=1015.581,9.904,-109.895,165.894,57.273,160.323
C01145=1015.574,9.554,-109.876,165.891,57.285,160.324
C01146=1015.568,9.304,-109.863,165.888,57.294,160.325
C01147=1015.563,9.055,-109.851,165.886,57.302,160.326
C01148=1015.558,8.805,-109.837,165.883,57.310,160.327
C01149=1015.553,8.556,-109.824,165.881,57.319,160.329
C01150=1015.548,8.305,-109.811,165.878,57.327,160.329
C01151=1015.542,8.056,-109.798,165.876,57.335,160.330
C01152=1015.537,7.807,-109.785,165.873,57.344,160.331
C01153=1015.532,7.556,-109.772,165.871,57.352,160.332
C01154=1015.527,7.308,-109.758,165.868,57.361,160.333
C01155=1015.522,7.057,-109.745,165.866,57.369,160.335
C01156=1015.517,6.808,-109.733,165.863,57.377,160.335
C01157=1015.511,6.558,-109.720,165.860,57.386,160.336
C01158=1015.506,6.309,-109.706,165.858,57.394,160.337
C01159=1015.501,6.059,-109.693,165.855,57.403,160.338
C01160=1015.496,5.810,-109.681,165.854,57.411,160.339
C01161=1015.491,5.560,-109.667,165.850,57.419,160.340
C01162=1015.487,5.346,-109.657,165.849,57.427,160.341
C01163=1015.482,5.131,-109.645,165.846,57.434,160.342
C01164=1015.478,4.915,-109.634,165.845,57.441,160.343
C01165=1015.473,4.701,-109.623,165.842,57.448,160.343
C01166=1015.469,4.486,-109.612,165.840,57.456,160.344
C01167=1015.464,4.272,-109.601,165.838,57.462,160.345
C01168=1015.460,4.057,-109.589,165.835,57.469,160.346
C01169=1015.456,3.841,-109.578,165.834,57.476,160.347
C01170=1015.450,3.592,-109.566,165.831,57.485,160.348
C01171=1015.445,3.342,-109.553,165.829,57.493,160.349
C01172=1015.440,3.093,-109.539,165.826,57.501,160.349
C01173=1015.435,2.843,-109.526,165.824,57.510,160.351
C01174=1015.430,2.594,-109.514,165.821,57.518,160.351
C01175=1015.425,2.344,-109.501,165.819,57.526,160.353
C01176=1015.420,2.094,-109.488,165.817,57.534,160.353
C01177=1015.415,1.845,-109.474,165.814,57.543,160.354
C01178=1015.409,1.595,-109.462,165.812,57.551,160.355
C01179=1015.405,1.346,-109.449,165.808,57.559,160.356
C01180=1015.400,1.096,-109.436,165.807,57.567,160.357
C01181=1015.395,0.846,-109.423,165.803,57.575,160.358
C01182=1015.390,0.597,-109.411,165.802,57.584,160.359
C01183=1015.385,0.347,-109.398,165.799,57.592,160.360
C01184=1015.380,0.098,-109.384,165.796,57.600,160.361
C01185=1015.374,-0.152,-109.371,165.794,57.608,160.362
C01186=1015.369,-0.402,-109.359,165.791,57.616,160.363
C01187=1015.365,-0.651,-109.346,165.789,57.624,160.364
C01188=1015.359,-0.901,-109.333,165.787,57.633,160.365
C01189=1015.354,-1.150,-109.321,165.784,57.641,160.365
C01190=1015.349,-1.401,-109.308,165.782,57.649,160.366
C01191=1015.344,-1.650,-109.295,165.778,57.657,160.367
C01192=1015.340,-1.900,-109.282,165.777,57.665,160.368
C01193=1015.334,-2.149,-109.270,165.774,57.673,160.369
C01194=1015.329,-2.398,-109.256,165.771,57.681,160.370
C01195=1015.324,-2.648,-109.243,165.769,57.689,160.371
C01196=1015.319,-2.898,-109.230,165.767,57.697,160.372
C01197=1015.314,-3.147,-109.218,165.764,57.706,160.373
C01198=1015.309,-3.397,-109.205,165.762,57.713,160.374
C01199=1015.304,-3.647,-109.192,165.758,57.722,160.374
C01200=1015.300,-3.896,-109.179,165.757,57.730,160.376
C01201=1015.294,-4.146,-109.167,165.755,57.738,160.376
C01202=1015.289,-4.396,-109.154,165.751,57.746,160.377
C01203=1015.285,-4.645,-109.141,165.749,57.754,160.378
C01204=1015.279,-4.896,-109.129,165.747,57.762,160.379
C01205=1015.274,-5.145,-109.117,165.744,57.770,160.380
C01206=1015.268,-5.423,-109.103,165.741,57.779,160.381
C01207=1015.262,-5.701,-109.089,165.739,57.789,160.382
C01208=1015.256,-5.979,-109.076,165.736,57.798,160.383
C01209=1015.251,-6.256,-109.062,165.733,57.807,160.384
C01210=1015.246,-6.507,-109.049,165.731,57.815,160.385
C01211=1015.241,-6.756,-109.037,165.728,57.824,160.386
C01212=1015.236,-7.006,-109.025,165.726,57.832,160.387
C01213=1015.231,-7.255,-109.012,165.723,57.840,160.388
C01214=1015.225,-7.505,-109.000,165.721,57.848,160.389
C01215=1015.220,-7.754,-108.988,165.718,57.857,160.390
C01216=1015.215,-8.004,-108.975,165.715,57.864,160.391
C01217=1015.210,-8.254,-108.963,165.713,57.873,160.392
C01218=1015.204,-8.503,-108.951,165.711,57.881,160.392
C01219=1015.200,-8.753,-108.938,165.707,57.889,160.393
C01220=1015.195,-9.003,-108.926,165.706,57.898,160.394
C01221=1015.189,-9.252,-108.914,165.704,57.906,160.395
C01222=1015.184,-9.502,-108.901,165.700,57.914,160.396
C01223=1015.179,-9.752,-108.890,165.698,57.922,160.397
C01224=1015.175,-10.001,-108.877,165.695,57.930,160.398
C01225=1015.169,-10.251,-108.865,165.693,57.938,160.399
C01226=1015.164,-10.501,-108.853,165.691,57.946,160.400
C01227=1015.159,-10.751,-108.840,165.688,57.954,160.400
C01228=1015.154,-11.000,-108.828,165.686,57.962,160.401
C01229=1015.149,-11.250,-108.816,165.682,57.970,160.402
C01230=1015.144,-11.499,-108.804,165.681,57.979,160.403
C01231=1015.138,-11.749,-108.791,165.679,57.987,160.404
C01232=1015.133,-11.999,-108.780,165.675,57.995,160.405
C01233=1015.129,-12.248,-108.767,165.673,58.003,160.406
C01234=1015.124,-12.497,-108.755,165.670,58.011,160.407
C01235=1015.119,-12.747,-108.743,165.668,58.019,160.408
C01236=1015.113,-12.997,-108.730,165.666,58.026,160.408
C01237=1015.108,-13.247,-108.719,165.662,58.035,160.409
C01238=1015.103,-13.496,-108.706,165.661,58.043,160.410
C01239=1015.098,-13.746,-108.694,165.659,58.051,160.411
C01240=1015.093,-13.996,-108.682,165.655,58.059,160.412
C01241=1015.089,-14.245,-108.669,165.653,58.067,160.413
C01242=1015.083,-14.496,-108.657,165.651,58.075,160.414
C01243=1015.078,-14.745,-108.645,165.648,58.083,160.415
C01244=1015.073,-14.994,-108.633,165.646,58.091,160.415
C01245=1015.068,-15.244,-108.621,165.643,58.099,160.416
C01246=1015.063,-15.493,-108.609,165.640,58.107,160.417
C01247=1015.059,-15.743,-108.597,165.638,58.115,160.418
C01248=1015.053,-15.993,-108.584,165.636,58.122,160.419
C01249=1015.048,-16.243,-108.573,165.633,58.131,160.420
C01250=1015.043,-16.493,-108.561,165.630,58.138,160.421
C01251=1015.038,-16.742,-108.549,165.628,58.146,160.421
C01252=1015.033,-16.992,-108.537,165.625,58.154,160.422
C01253=1015.028,-17.241,-108.525,165.623,58.162,160.423
C01254=1015.023,-17.491,-108.513,165.620,58.170,160.424
C01255=1015.018,-17.741,-108.502,165.618,58.179,160.425
C01256=1015.012,-17.991,-108.489,165.616,58.187,160.426
C01257=1015.007,-18.241,-108.478,165.613,58.195,160.427
C01258=1015.002,-18.490,-108.466,165.611,58.203,160.428
C01259=1014.997,-18.740,-108.454,165.607,58.211,160.428
C01260=1014.992,-18.989,-108.443,165.605,58.219,160.429
C01261=1014.987,-19.239,-108.431,165.603,58.227,160.430
C01262=1014.982,-19.488,-108.419,165.600,58.235,160.431
C01263=1014.977,-19.738,-108.408,165.598,58.243,160.432
C01264=1014.972,-19.988,-108.396,165.596,58.251,160.433
C01265=1014.966,-20.237,-108.384,165.592,58.259,160.433
C01266=1014.961,-20.487,-108.372,165.590,58.267,160.434
C01267=1014.957,-20.737,-108.360,165.588,58.275,160.435
C01268=1014.952,-20.987,-108.349,165.585,58.283,160.436
C01269=1014.947,-21.236,-108.337,165.583,58.291,160.437
C01270=1014.940,-21.513,-108.325,165.580,58.300,160.438
C01271=1014.935,-21.789,-108.311,165.577,58.308,160.439
C01272=1014.930,-22.065,-108.298,165.575,58.317,160.440
C01273=1014.924,-22.342,-108.285,165.571,58.325,160.440
C01274=1014.919,-22.591,-108.273,165.569,58.333,160.441
C01275=1014.914,-22.840,-108.262,165.566,58.341,160.442
C01276=1014.909,-23.090,-108.250,165.564,58.349,160.443
C01277=1014.904,-23.340,-108.239,165.562,58.357,160.444
C01278=1014.899,-23.589,-108.227,165.559,58.365,160.445
C01279=1014.894,-23.839,-108.215,165.556,58.373,160.446
C01280=1014.889,-24.089,-108.204,165.554,58.380,160.446
C01281=1014.884,-24.339,-108.192,165.552,58.388,160.447
C01282=1014.879,-24.588,-108.181,165.548,58.396,160.448
C01283=1014.873,-24.838,-108.169,165.546,58.404,160.449
C01284=1014.868,-25.087,-108.157,165.544,58.412,160.450
C01285=1014.863,-25.337,-108.146,165.542,58.419,160.450
C01286=1014.858,-25.587,-108.134,165.538,58.427,160.451
C01287=1014.854,-25.837,-108.122,165.536,58.435,160.452
C01288=1014.850,-26.086,-108.111,165.534,58.443,160.453
C01289=1014.845,-26.336,-108.100,165.531,58.450,160.453
C01290=1014.839,-26.585,-108.087,165.529,58.458,160.454
C01291=1014.834,-26.835,-108.076,165.526,58.466,160.455
C01292=1014.829,-27.085,-108.064,165.523,58.473,160.456
C01293=1014.824,-27.335,-108.053,165.521,58.481,160.457
C01294=1014.819,-27.584,-108.041,165.519,58.489,160.458
C01295=1014.814,-27.834,-108.030,165.517,58.497,160.459
C01296=1014.809,-28.084,-108.018,165.513,58.504,160.459
C01297=1014.804,-28.334,-108.007,165.511,58.512,160.460
C01298=1014.799,-28.583,-107.996,165.509,58.520,160.461
C01299=1014.794,-28.833,-107.985,165.506,58.528,160.461
C01300=1014.789,-29.083,-107.973,165.504,58.536,160.462
C01301=1014.784,-29.332,-107.962,165.501,58.543,160.463
C01302=1014.778,-29.582,-107.951,165.498,58.551,160.464
C01303=1014.773,-29.831,-107.940,165.496,58.559,160.465
C01304=1014.769,-30.082,-107.929,165.494,58.567,160.466
C01305=1014.764,-30.332,-107.918,165.492,58.575,160.467
C01306=1014.758,-30.581,-107.907,165.488,58.583,160.467
C01307=1014.753,-30.831,-107.895,165.486,58.590,160.468
C01308=1014.749,-31.080,-107.884,165.484,58.598,160.469
C01309=1014.744,-31.330,-107.873,165.481,58.605,160.469
C01310=1014.739,-31.580,-107.861,165.478,58.614,160.470
C01311=1014.733,-31.829,-107.850,165.476,58.622,160.471
C01312=1014.728,-32.079,-107.839,165.474,58.629,160.472
C01313=1014.723,-32.329,-107.828,165.471,58.637,160.473
C01314=1014.719,-32.578,-107.817,165.468,58.645,160.473
C01315=1014.713,-32.828,-107.806,165.466,58.653,160.474
C01316=1014.708,-33.078,-107.795,165.463,58.660,160.475
C01317=1014.703,-33.327,-107.783,165.461,58.668,160.476
C01318=1014.698,-33.578,-107.772,165.459,58.675,160.476
C01319=1014.693,-33.827,-107.762,165.455,58.683,160.477
C01320=1014.688,-34.076,-107.750,165.453,58.691,160.478
C01321=1014.683,-34.326,-107.739,165.451,58.698,160.479
C01322=1014.678,-34.576,-107.727,165.449,58.706,160.480
C01323=1014.673,-34.826,-107.717,165.446,58.713,160.480
C01324=1014.668,-35.075,-107.706,165.443,58.721,160.481
C01325=1014.663,-35.325,-107.695,165.440,58.729,160.482
C01326=1014.658,-35.575,-107.683,165.438,58.736,160.483
C01327=1014.653,-35.825,-107.673,165.435,58.744,160.483
C01328=1014.649,-36.074,-107.662,165.433,58.751,160.484
C01329=1014.644,-36.324,-107.650,165.431,58.759,160.485
C01330=1014.639,-36.574,-107.639,165.429,58.766,160.486
C01331=1014.633,-36.824,-107.629,165.425,58.774,160.486
C01332=1014.629,-37.073,-107.618,165.423,58.782,160.487
C01333=1014.624,-37.323,-107.606,165.420,58.789,160.488
C01334=1014.618,-37.598,-107.594,165.417,58.797,160.488
C01335=1014.613,-37.873,-107.582,165.415,58.805,160.489
C01336=1014.607,-38.148,-107.570,165.412,58.814,160.490
C01337=1014.602,-38.423,-107.558,165.409,58.822,160.491
C01338=1014.597,-38.673,-107.547,165.407,58.830,160.492
C01339=1014.592,-38.923,-107.536,165.404,58.837,160.492
C01340=1014.587,-39.172,-107.525,165.401,58.844,160.493
C01341=1014.582,-39.422,-107.514,165.399,58.852,160.494
C01342=1014.577,-39.672,-107.503,165.397,58.859,160.494
C01343=1014.572,-39.922,-107.493,165.395,58.867,160.495
C01344=1014.567,-40.171,-107.482,165.392,58.874,160.496
C01345=1014.562,-40.422,-107.471,165.389,58.882,160.497
C01346=1014.558,-40.671,-107.460,165.386,58.890,160.497
C01347=1014.552,-40.921,-107.450,165.384,58.897,160.498
C01348=1014.547,-41.171,-107.439,165.382,58.905,160.499
C01349=1014.542,-41.420,-107.429,165.379,58.912,160.500
C01350=1014.537,-41.670,-107.417,165.377,58.920,160.500
C01351=1014.532,-41.920,-107.407,165.374,58.927,160.501
C01352=1014.527,-42.169,-107.396,165.371,58.935,160.502
C01353=1014.522,-42.419,-107.386,165.369,58.942,160.502
C01354=1014.518,-42.668,-107.375,165.366,58.949,160.503
C01355=1014.512,-42.918,-107.365,165.364,58.957,160.504
C01356=1014.508,-43.169,-107.354,165.361,58.965,160.505
C01357=1014.502,-43.417,-107.343,165.359,58.972,160.506
C01358=1014.497,-43.668,-107.333,165.357,58.980,160.506
C01359=1014.493,-43.917,-107.322,165.354,58.987,160.507
C01360=1014.487,-44.167,-107.312,165.351,58.994,160.507
C01361=1014.482,-44.417,-107.301,165.349,59.002,160.508
C01362=1014.477,-44.666,-107.291,165.346,59.009,160.509
///RCONF 1,0,0,1,0,0,0,0,0,0,0,0,0,0,0,0,0,0,0,0,0,0,0,0
C01363=1014.473,-44.916,-107.280,165.343,59.017,160.509
C01364=1014.467,-45.165,-107.269,165.341,59.024,160.510
C01365=1014.463,-45.416,-107.259,165.338,59.032,160.511
C01366=1014.457,-45.666,-107.249,165.336,59.039,160.512
C01367=1014.453,-45.915,-107.237,165.333,59.046,160.512
C01368=1014.447,-46.165,-107.227,165.331,59.054,160.513
C01369=1014.443,-46.415,-107.217,165.328,59.061,160.514
C01370=1014.438,-46.664,-107.206,165.326,59.068,160.514
C01371=1014.434,-46.914,-107.196,165.323,59.075,160.515
C01372=1014.428,-47.164,-107.185,165.321,59.083,160.516
C01373=1014.423,-47.413,-107.175,165.318,59.090,160.516
C01374=1014.418,-47.663,-107.164,165.316,59.098,160.517
C01375=1014.413,-47.913,-107.154,165.313,59.105,160.518
C01376=1014.408,-48.162,-107.143,165.311,59.112,160.518
C01377=1014.404,-48.412,-107.133,165.308,59.119,160.519
C01378=1014.399,-48.662,-107.122,165.305,59.126,160.520
C01379=1014.394,-48.912,-107.113,165.303,59.134,160.520
C01380=1014.389,-49.161,-107.101,165.300,59.141,160.521
C01381=1014.384,-49.411,-107.091,165.298,59.148,160.521
C01382=1014.380,-49.661,-107.081,165.296,59.155,160.522
C01383=1014.375,-49.911,-107.071,165.293,59.162,160.523
C01384=1014.370,-50.160,-107.059,165.291,59.169,160.524
C01385=1014.365,-50.410,-107.049,165.288,59.176,160.524
C01386=1014.359,-50.660,-107.039,165.286,59.183,160.525
C01387=1014.355,-50.910,-107.029,165.283,59.190,160.525
C01388=1014.350,-51.160,-107.019,165.280,59.198,160.526
C01389=1014.346,-51.410,-107.008,165.278,59.205,160.527
C01390=1014.340,-51.660,-106.998,165.276,59.213,160.528
C01391=1014.336,-51.909,-106.988,165.273,59.220,160.528
C01392=1014.330,-52.159,-106.978,165.271,59.227,160.529
C01393=1014.325,-52.409,-106.968,165.268,59.234,160.529
C01394=1014.320,-52.659,-106.958,165.265,59.242,160.530
C01395=1014.315,-52.908,-106.949,165.263,59.249,160.531
C01396=1014.310,-53.158,-106.939,165.261,59.257,160.532
C01397=1014.305,-53.408,-106.929,165.258,59.264,160.532
C01398=1014.299,-53.682,-106.918,165.255,59.272,160.533
C01399=1014.294,-53.958,-106.906,165.251,59.280,160.533
C01400=1014.288,-54.234,-106.896,165.249,59.288,160.534
C01401=1014.283,-54.509,-106.885,165.246,59.296,160.535
C01402=1014.278,-54.759,-106.874,165.244,59.303,160.536
C01403=1014.273,-55.009,-106.865,165.241,59.311,160.536
C01404=1014.268,-55.258,-106.855,165.239,59.318,160.537
C01405=1014.263,-55.508,-106.845,165.236,59.325,160.538
C01406=1014.258,-55.758,-106.836,165.233,59.332,160.538
C01407=1014.253,-56.008,-106.826,165.231,59.339,160.539
C01408=1014.248,-56.258,-106.816,165.228,59.347,160.539
C01409=1014.243,-56.507,-106.806,165.226,59.354,160.540
C01410=1014.238,-56.756,-106.796,165.223,59.361,160.541
C01411=1014.233,-57.007,-106.786,165.220,59.368,160.541
C01412=1014.228,-57.256,-106.776,165.218,59.375,160.542
C01413=1014.223,-57.506,-106.767,165.215,59.383,160.543
C01414=1014.218,-57.756,-106.757,165.214,59.389,160.543
C01415=1014.213,-58.005,-106.747,165.211,59.397,160.544
C01416=1014.208,-58.255,-106.737,165.209,59.404,160.545
C01417=1014.203,-58.505,-106.727,165.206,59.411,160.545
C01418=1014.198,-58.755,-106.718,165.203,59.418,160.546
C01419=1014.194,-59.004,-106.708,165.201,59.425,160.547
C01420=1014.188,-59.255,-106.698,165.198,59.432,160.547
C01421=1014.183,-59.504,-106.688,165.195,59.439,160.547
C01422=1014.178,-59.753,-106.678,165.194,59.446,160.548
C01423=1014.174,-60.003,-106.669,165.191,59.453,160.549
C01424=1014.169,-60.254,-106.659,165.188,59.460,160.550
C01425=1014.164,-60.503,-106.649,165.185,59.467,160.550
C01426=1014.160,-60.753,-106.639,165.183,59.474,160.550
C01427=1014.155,-61.003,-106.630,165.180,59.481,160.551
C01428=1014.150,-61.253,-106.620,165.179,59.488,160.552
C01429=1014.145,-61.502,-106.610,165.175,59.494,160.552
C01430=1014.140,-61.752,-106.600,165.173,59.502,160.553
C01431=1014.135,-62.002,-106.591,165.170,59.509,160.553
C01432=1014.130,-62.252,-106.581,165.168,59.516,160.554
C01433=1014.125,-62.501,-106.571,165.165,59.522,160.555
C01434=1014.121,-62.751,-106.562,165.163,59.529,160.555
C01435=1014.116,-63.001,-106.552,165.160,59.536,160.556
C01436=1014.110,-63.251,-106.542,165.157,59.543,160.556
C01437=1014.106,-63.501,-106.533,165.156,59.550,160.557
C01438=1014.101,-63.750,-106.523,165.153,59.557,160.558
C01439=1014.096,-64.000,-106.513,165.150,59.563,160.558
C01440=1014.092,-64.250,-106.504,165.147,59.571,160.558
C01441=1014.086,-64.500,-106.494,165.145,59.577,160.559
C01442=1014.081,-64.749,-106.484,165.143,59.584,160.560
C01443=1014.077,-64.999,-106.475,165.139,59.590,160.560
C01444=1014.072,-65.248,-106.466,165.138,59.597,160.561
C01445=1014.067,-65.498,-106.456,165.135,59.604,160.561
C01446=1014.063,-65.748,-106.447,165.132,59.611,160.562
C01447=1014.057,-65.998,-106.436,165.131,59.618,160.563
C01448=1014.053,-66.248,-106.427,165.127,59.624,160.563
C01449=1014.048,-66.497,-106.418,165.125,59.631,160.563
C01450=1014.043,-66.747,-106.408,165.123,59.637,160.564
C01451=1014.039,-66.997,-106.399,165.120,59.644,160.564
C01452=1014.034,-67.246,-106.389,165.117,59.651,160.565
C01453=1014.029,-67.496,-106.380,165.115,59.657,160.565
C01454=1014.024,-67.746,-106.370,165.112,59.664,160.566
C01455=1014.019,-67.996,-106.361,165.110,59.670,160.566
C01456=1014.014,-68.246,-106.351,165.108,59.677,160.567
C01457=1014.010,-68.495,-106.341,165.104,59.684,160.567
C01458=1014.005,-68.745,-106.332,165.102,59.690,160.568
C01459=1014.000,-68.995,-106.322,165.100,59.697,160.569
C01460=1013.996,-69.245,-106.313,165.098,59.703,160.569
C01461=1013.991,-69.494,-106.303,165.094,59.710,160.569
C01462=1013.986,-69.771,-106.293,165.092,59.717,160.570
C01463=1013.981,-70.048,-106.282,165.089,59.724,160.571
C01464=1013.975,-70.323,-106.272,165.087,59.731,160.571
C01465=1013.970,-70.600,-106.262,165.084,59.739,160.572
C01466=1013.965,-70.850,-106.252,165.081,59.745,160.572
C01467=1013.961,-71.100,-106.243,165.079,59.751,160.573
C01468=1013.956,-71.349,-106.233,165.076,59.758,160.573
C01469=1013.952,-71.599,-106.224,165.074,59.765,160.574
C01470=1013.947,-71.849,-106.214,165.071,59.771,160.574
C01471=1013.942,-72.099,-106.205,165.069,59.777,160.575
C01472=1013.937,-72.348,-106.195,165.066,59.784,160.575
C01473=1013.933,-72.598,-106.186,165.064,59.790,160.575
C01474=1013.928,-72.848,-106.177,165.060,59.796,160.576
C01475=1013.924,-73.098,-106.167,165.059,59.803,160.577
C01476=1013.919,-73.348,-106.158,165.056,59.809,160.577
C01477=1013.914,-73.597,-106.148,165.054,59.815,160.577
C01478=1013.910,-73.847,-106.139,165.051,59.822,160.578
C01479=1013.905,-74.096,-106.129,165.048,59.828,160.578
C01480=1013.900,-74.347,-106.120,165.046,59.834,160.579
C01481=1013.896,-74.597,-106.111,165.043,59.841,160.579
C01482=1013.891,-74.846,-106.101,165.041,59.847,160.579
C01483=1013.886,-75.096,-106.092,165.038,59.853,160.580
C01484=1013.881,-75.346,-106.084,165.036,59.860,160.581
C01485=1013.877,-75.596,-106.075,165.033,59.866,160.581
C01486=1013.872,-75.846,-106.066,165.031,59.872,160.581
C01487=1013.867,-76.095,-106.057,165.028,59.879,160.582
C01488=1013.862,-76.345,-106.047,165.026,59.885,160.582
C01489=1013.857,-76.595,-106.038,165.023,59.892,160.583
C01490=1013.853,-76.845,-106.029,165.021,59.898,160.583
C01491=1013.848,-77.095,-106.021,165.018,59.905,160.584
C01492=1013.843,-77.345,-106.012,165.016,59.911,160.584
C01493=1013.839,-77.595,-106.003,165.013,59.917,160.584
C01494=1013.833,-77.844,-105.993,165.011,59.923,160.585
C01495=1013.829,-78.093,-105.985,165.009,59.929,160.585
C01496=1013.825,-78.343,-105.976,165.005,59.936,160.586
C01497=1013.819,-78.593,-105.967,165.003,59.942,160.586
C01498=1013.815,-78.843,-105.958,165.000,59.949,160.586
C01499=1013.810,-79.093,-105.949,164.998,59.955,160.587
C01500=1013.805,-79.343,-105.940,164.996,59.961,160.588
C01501=1013.800,-79.593,-105.931,164.993,59.967,160.588
C01502=1013.796,-79.843,-105.922,164.991,59.973,160.588
C01503=1013.791,-80.093,-105.913,164.987,59.980,160.589
C01504=1013.786,-80.342,-105.905,164.985,59.986,160.589
C01505=1013.782,-80.592,-105.896,164.983,59.992,160.590
C01506=1013.777,-80.841,-105.888,164.980,59.998,160.590
C01507=1013.772,-81.091,-105.878,164.979,60.005,160.591
C01508=1013.767,-81.341,-105.870,164.976,60.012,160.591
C01509=1013.763,-81.591,-105.861,164.973,60.018,160.592
C01510=1013.757,-81.841,-105.852,164.970,60.024,160.592
C01511=1013.753,-82.090,-105.844,164.968,60.030,160.592
C01512=1013.748,-82.340,-105.835,164.966,60.036,160.593
C01513=1013.743,-82.590,-105.827,164.963,60.043,160.593
C01514=1013.739,-82.840,-105.818,164.961,60.049,160.594
C01515=1013.733,-83.090,-105.810,164.958,60.056,160.594
C01516=1013.730,-83.339,-105.801,164.956,60.062,160.594
C01517=1013.724,-83.589,-105.793,164.953,60.068,160.595
C01518=1013.719,-83.839,-105.784,164.950,60.074,160.595
C01519=1013.715,-84.089,-105.776,164.948,60.080,160.596
C01520=1013.710,-84.339,-105.767,164.946,60.086,160.596
C01521=1013.706,-84.589,-105.759,164.943,60.093,160.597
C01522=1013.700,-84.838,-105.750,164.940,60.098,160.597
C01523=1013.695,-85.088,-105.742,164.938,60.104,160.597
C01524=1013.691,-85.339,-105.733,164.935,60.111,160.598
C01525=1013.686,-85.588,-105.725,164.933,60.117,160.598
C01526=1013.681,-85.866,-105.715,164.930,60.123,160.598
C01527=1013.675,-86.144,-105.706,164.927,60.131,160.599
C01528=1013.670,-86.423,-105.697,164.924,60.137,160.599
C01529=1013.665,-86.701,-105.687,164.923,60.144,160.600
C01530=1013.660,-86.951,-105.679,164.919,60.150,160.600
C01531=1013.655,-87.201,-105.670,164.917,60.156,160.601
C01532=1013.651,-87.451,-105.662,164.915,60.162,160.601
C01533=1013.646,-87.700,-105.654,164.913,60.168,160.602
C01534=1013.642,-87.950,-105.644,164.909,60.174,160.601
C01535=1013.637,-88.200,-105.637,164.907,60.180,160.602
C01536=1013.632,-88.450,-105.629,164.905,60.186,160.603
C01537=1013.627,-88.700,-105.619,164.902,60.191,160.603
C01538=1013.622,-88.950,-105.612,164.900,60.197,160.603
C01539=1013.618,-89.199,-105.603,164.897,60.204,160.603
C01540=1013.613,-89.449,-105.595,164.894,60.209,160.604
C01541=1013.609,-89.700,-105.586,164.892,60.215,160.604
C01542=1013.604,-89.949,-105.578,164.890,60.221,160.605
C01543=1013.599,-90.198,-105.570,164.887,60.227,160.605
C01544=1013.595,-90.448,-105.562,164.885,60.233,160.605
C01545=1013.590,-90.698,-105.553,164.882,60.238,160.606
C01546=1013.586,-90.948,-105.544,164.880,60.244,160.606
C01547=1013.581,-91.198,-105.537,164.876,60.250,160.606
C01548=1013.576,-91.447,-105.528,164.874,60.256,160.606
C01549=1013.572,-91.697,-105.519,164.872,60.261,160.607
C01550=1013.567,-91.947,-105.512,164.870,60.268,160.607
C01551=1013.563,-92.197,-105.503,164.867,60.273,160.607
C01552=1013.558,-92.447,-105.495,164.865,60.279,160.608
C01553=1013.553,-92.696,-105.487,164.862,60.284,160.608
C01554=1013.548,-92.946,-105.478,164.860,60.290,160.609
C01555=1013.544,-93.196,-105.470,164.857,60.296,160.609
C01556=1013.539,-93.446,-105.462,164.855,60.302,160.609
C01557=1013.535,-93.696,-105.454,164.852,60.307,160.609
C01558=1013.530,-93.945,-105.445,164.850,60.312,160.610
C01559=1013.526,-94.196,-105.437,164.848,60.319,160.610
C01560=1013.521,-94.445,-105.429,164.845,60.324,160.610
C01561=1013.516,-94.695,-105.420,164.842,60.329,160.610
C01562=1013.512,-94.945,-105.412,164.840,60.335,160.611
C01563=1013.507,-95.195,-105.404,164.837,60.341,160.611
C01564=1013.503,-95.444,-105.396,164.835,60.346,160.611
C01565=1013.498,-95.694,-105.387,164.833,60.352,160.612
C01566=1013.494,-95.944,-105.380,164.830,60.357,160.612
C01567=1013.489,-96.194,-105.371,164.827,60.363,160.612
C01568=1013.485,-96.443,-105.363,164.825,60.368,160.612
C01569=1013.480,-96.694,-105.354,164.823,60.374,160.613
C01570=1013.475,-96.944,-105.347,164.821,60.379,160.613
C01571=1013.471,-97.193,-105.338,164.818,60.384,160.613
C01572=1013.466,-97.444,-105.330,164.815,60.390,160.613
C01573=1013.462,-97.693,-105.323,164.812,60.395,160.614
C01574=1013.458,-97.943,-105.314,164.810,60.401,160.614
C01575=1013.453,-98.193,-105.306,164.809,60.406,160.615
C01576=1013.448,-98.443,-105.298,164.806,60.411,160.615
C01577=1013.444,-98.692,-105.290,164.803,60.417,160.615
C01578=1013.439,-98.942,-105.283,164.801,60.423,160.615
C01579=1013.434,-99.192,-105.275,164.799,60.428,160.616
C01580=1013.430,-99.441,-105.267,164.796,60.434,160.616
C01581=1013.425,-99.691,-105.259,164.793,60.439,160.616
C01582=1013.421,-99.941,-105.251,164.791,60.445,160.616
C01583=1013.416,-100.192,-105.243,164.788,60.450,160.617
C01584=1013.411,-100.441,-105.235,164.786,60.456,160.617
C01585=1013.406,-100.691,-105.228,164.783,60.461,160.617
C01586=1013.402,-100.941,-105.220,164.781,60.466,160.617
C01587=1013.397,-101.191,-105.212,164.779,60.471,160.617
C01588=1013.393,-101.441,-105.205,164.776,60.477,160.618
C01589=1013.388,-101.690,-105.197,164.774,60.483,160.618
C01590=1013.383,-101.970,-105.188,164.771,60.488,160.618
C01591=1013.378,-102.251,-105.180,164.768,60.495,160.619
C01592=1013.373,-102.532,-105.171,164.765,60.500,160.619
C01593=1013.368,-102.811,-105.162,164.763,60.506,160.619
C01594=1013.363,-103.062,-105.155,164.760,60.511,160.619
C01595=1013.359,-103.311,-105.146,164.758,60.517,160.620
C01596=1013.354,-103.561,-105.139,164.755,60.522,160.620
C01597=1013.349,-103.811,-105.131,164.753,60.527,160.620
C01598=1013.345,-104.060,-105.124,164.751,60.532,160.620
C01599=1013.340,-104.311,-105.116,164.748,60.538,160.620
C01600=1013.336,-104.560,-105.109,164.745,60.543,160.621
C01601=1013.331,-104.810,-105.101,164.744,60.548,160.621
C01602=1013.327,-105.061,-105.093,164.741,60.553,160.621
C01603=1013.322,-105.310,-105.085,164.738,60.559,160.621
C01604=1013.318,-105.559,-105.077,164.736,60.564,160.622
C01605=1013.313,-105.810,-105.070,164.734,60.569,160.622
C01606=1013.309,-106.059,-105.062,164.731,60.574,160.622
C01607=1013.304,-106.309,-105.055,164.729,60.578,160.622
C01608=1013.299,-106.559,-105.047,164.726,60.584,160.622
C01609=1013.295,-106.809,-105.040,164.723,60.589,160.622
C01610=1013.291,-107.058,-105.032,164.722,60.594,160.623
C01611=1013.286,-107.309,-105.024,164.719,60.599,160.623
C01612=1013.281,-107.558,-105.017,164.716,60.605,160.623
C01613=1013.277,-107.808,-105.010,164.714,60.609,160.623
C01614=1013.273,-108.058,-105.002,164.711,60.614,160.623
C01615=1013.268,-108.308,-104.994,164.710,60.619,160.624
C01616=1013.263,-108.558,-104.987,164.707,60.625,160.624
C01617=1013.259,-108.807,-104.980,164.704,60.630,160.624
C01618=1013.255,-109.057,-104.972,164.703,60.635,160.624
C01619=1013.250,-109.308,-104.965,164.699,60.639,160.624
C01620=1013.245,-109.557,-104.958,164.697,60.644,160.625
C01621=1013.240,-109.807,-104.951,164.695,60.650,160.625
C01622=1013.236,-110.056,-104.944,164.692,60.655,160.625
C01623=1013.231,-110.307,-104.936,164.690,60.659,160.625
C01624=1013.227,-110.556,-104.928,164.687,60.665,160.625
C01625=1013.222,-110.806,-104.921,164.685,60.669,160.626
C01626=1013.218,-111.056,-104.914,164.683,60.675,160.626
C01627=1013.213,-111.307,-104.907,164.680,60.679,160.626
C01628=1013.209,-111.556,-104.899,164.678,60.684,160.626
C01629=1013.205,-111.806,-104.892,164.676,60.689,160.626
C01630=1013.200,-112.055,-104.885,164.673,60.694,160.626
C01631=1013.195,-112.305,-104.878,164.671,60.699,160.627
C01632=1013.191,-112.556,-104.870,164.668,60.703,160.626
C01633=1013.186,-112.805,-104.863,164.666,60.708,160.627
C01634=1013.182,-113.055,-104.856,164.663,60.714,160.627
C01635=1013.178,-113.305,-104.848,164.661,60.718,160.627
C01636=1013.173,-113.554,-104.841,164.659,60.723,160.627
C01637=1013.169,-113.805,-104.834,164.656,60.727,160.627
C01638=1013.163,-114.055,-104.827,164.654,60.732,160.628
C01639=1013.159,-114.304,-104.820,164.651,60.737,160.627
C01640=1013.155,-114.554,-104.812,164.649,60.742,160.628
C01641=1013.151,-114.804,-104.806,164.647,60.746,160.628
C01642=1013.146,-115.054,-104.798,164.644,60.751,160.628
C01643=1013.142,-115.303,-104.791,164.642,60.755,160.628
C01644=1013.137,-115.554,-104.784,164.640,60.760,160.628
C01645=1013.132,-115.804,-104.777,164.637,60.765,160.628
C01646=1013.128,-116.053,-104.769,164.635,60.770,160.629
C01647=1013.124,-116.304,-104.763,164.632,60.774,160.628
C01648=1013.119,-116.553,-104.755,164.630,60.779,160.628
C01649=1013.114,-116.803,-104.749,164.628,60.783,160.629
C01650=1013.110,-117.053,-104.742,164.625,60.788,160.629
C01651=1013.106,-117.302,-104.734,164.623,60.793,160.629
C01652=1013.102,-117.552,-104.727,164.621,60.797,160.629
C01653=1013.097,-117.802,-104.721,164.618,60.801,160.629
C01654=1013.092,-118.083,-104.713,164.616,60.807,160.629
C01655=1013.086,-118.364,-104.705,164.613,60.812,160.629
C01656=1013.082,-118.644,-104.697,164.610,60.817,160.630
C01657=1013.076,-118.925,-104.690,164.607,60.822,160.629
C01658=1013.072,-119.175,-104.682,164.605,60.827,160.630
C01659=1013.068,-119.424,-104.675,164.603,60.831,160.630
C01660=1013.064,-119.675,-104.668,164.601,60.835,160.630
C01661=1013.058,-119.924,-104.661,164.598,60.841,160.630
C01662=1013.054,-120.174,-104.655,164.596,60.845,160.630
C01663=1013.050,-120.424,-104.647,164.593,60.849,160.630
C01664=1013.045,-120.674,-104.641,164.591,60.853,160.630
C01665=1013.041,-120.923,-104.634,164.589,60.857,160.630
C01666=1013.037,-121.174,-104.627,164.587,60.862,160.631
C01667=1013.032,-121.423,-104.620,164.584,60.867,160.630
C01668=1013.028,-121.673,-104.614,164.581,60.871,160.630
C01669=1013.023,-121.923,-104.606,164.579,60.875,160.630
C01670=1013.019,-122.173,-104.600,164.577,60.879,160.631
C01671=1013.014,-122.423,-104.593,164.575,60.883,160.631
C01672=1013.010,-122.673,-104.586,164.572,60.888,160.631
C01673=1013.006,-122.923,-104.579,164.571,60.893,160.631
C01674=1013.001,-123.172,-104.573,164.568,60.897,160.631
C01675=1012.997,-123.422,-104.566,164.566,60.901,160.631
C01676=1012.993,-123.672,-104.558,164.563,60.905,160.631
C01677=1012.988,-123.922,-104.552,164.560,60.910,160.631
C01678=1012.984,-124.172,-104.546,164.558,60.914,160.631
C01679=1012.979,-124.422,-104.538,164.556,60.918,160.631
C01680=1012.975,-124.672,-104.532,164.553,60.922,160.631
C01681=1012.971,-124.922,-104.526,164.551,60.926,160.631
C01682=1012.965,-125.171,-104.519,164.549,60.930,160.631
C01683=1012.961,-125.422,-104.512,164.547,60.935,160.631
C01684=1012.957,-125.671,-104.506,164.544,60.939,160.631
C01685=1012.953,-125.920,-104.499,164.542,60.943,160.631
C01686=1012.949,-126.171,-104.492,164.540,60.947,160.631
C01687=1012.944,-126.421,-104.486,164.537,60.951,160.631
C01688=1012.940,-126.671,-104.479,164.535,60.955,160.631
C01689=1012.935,-126.920,-104.473,164.533,60.960,160.631
C01690=1012.931,-127.171,-104.466,164.530,60.964,160.631
C01691=1012.926,-127.420,-104.460,164.527,60.967,160.631
C01692=1012.922,-127.671,-104.453,164.525,60.971,160.631
C01693=1012.917,-127.919,-104.447,164.524,60.975,160.631
C01694=1012.913,-128.170,-104.440,164.522,60.979,160.632
C01695=1012.909,-128.418,-104.434,164.519,60.983,160.632
C01696=1012.905,-128.668,-104.426,164.516,60.987,160.631
C01697=1012.901,-128.918,-104.418,164.514,60.990,160.631
C01698=1012.898,-129.168,-104.410,164.513,60.993,160.631
C01699=1012.895,-129.417,-104.401,164.510,60.995,160.631
C01700=1012.893,-129.667,-104.391,164.508,60.996,160.630
C01701=1012.890,-129.916,-104.380,164.505,60.998,160.630
C01702=1012.888,-130.166,-104.369,164.504,61.000,160.630
C01703=1012.886,-130.415,-104.358,164.501,61.000,160.629
C01704=1012.885,-130.665,-104.346,164.500,61.000,160.628
C01705=1012.884,-130.915,-104.333,164.497,61.000,160.627
C01706=1012.884,-131.165,-104.319,164.495,61.000,160.627
C01707=1012.883,-131.414,-104.305,164.492,60.999,160.626
C01708=1012.883,-131.664,-104.291,164.492,60.998,160.625
C01709=1012.884,-131.914,-104.276,164.488,60.997,160.624
C01710=1012.885,-132.163,-104.260,164.487,60.995,160.623
C01711=1012.885,-132.413,-104.243,164.485,60.993,160.622
C01712=1012.886,-132.663,-104.226,164.483,60.990,160.621
C01713=1012.888,-132.913,-104.208,164.481,60.987,160.620
C01714=1012.890,-133.162,-104.190,164.479,60.983,160.619
C01715=1012.893,-133.412,-104.171,164.477,60.980,160.617
C01716=1012.895,-133.661,-104.152,164.475,60.976,160.616
C01717=1012.899,-133.910,-104.132,164.473,60.971,160.614
C01718=1012.843,-119.412,-105.099,164.589,61.092,160.675
C01719=1012.851,-119.017,-105.110,164.594,61.085,160.675
C01720=1012.858,-118.620,-105.121,164.597,61.079,160.675
C01721=1012.865,-118.225,-105.132,164.600,61.073,160.675
C01722=1012.872,-117.829,-105.143,164.605,61.066,160.675
C01723=1012.876,-117.579,-105.150,164.607,61.061,160.675
C01724=1012.880,-117.329,-105.158,164.609,61.057,160.675
C01725=1012.885,-117.080,-105.164,164.612,61.053,160.675
C01726=1012.890,-116.830,-105.171,164.614,61.049,160.675
C01727=1012.894,-116.580,-105.178,164.616,61.045,160.675
C01728=1012.898,-116.330,-105.185,164.618,61.041,160.675
C01729=1012.903,-116.080,-105.192,164.621,61.036,160.675
C01730=1012.907,-115.831,-105.199,164.623,61.032,160.675
C01731=1012.911,-115.580,-105.206,164.625,61.028,160.674
C01732=1012.916,-115.331,-105.213,164.628,61.024,160.674
C01733=1012.921,-115.082,-105.220,164.630,61.020,160.674
C01734=1012.926,-114.831,-105.227,164.632,61.016,160.674
C01735=1012.930,-114.581,-105.235,164.634,61.011,160.674
C01736=1012.934,-114.331,-105.242,164.638,61.007,160.674
C01737=1012.938,-114.081,-105.249,164.639,61.002,160.674
C01738=1012.943,-113.831,-105.256,164.642,60.998,160.674
C01739=1012.947,-113.582,-105.264,164.644,60.994,160.674
C01740=1012.951,-113.332,-105.271,164.646,60.989,160.674
C01741=1012.957,-113.082,-105.277,164.648,60.985,160.674
C01742=1012.961,-112.832,-105.285,164.651,60.981,160.674
C01743=1012.965,-112.582,-105.292,164.653,60.976,160.674
C01744=1012.970,-112.333,-105.300,164.656,60.972,160.674
C01745=1012.974,-112.082,-105.306,164.658,60.967,160.674
C01746=1012.978,-111.833,-105.314,164.660,60.963,160.673
C01747=1012.983,-111.583,-105.321,164.663,60.958,160.673
C01748=1012.988,-111.333,-105.329,164.665,60.954,160.673
C01749=1012.992,-111.083,-105.336,164.668,60.950,160.673
C01750=1012.997,-110.833,-105.342,164.669,60.945,160.673
C01751=1013.001,-110.584,-105.350,164.673,60.940,160.673
C01752=1013.005,-110.334,-105.357,164.675,60.936,160.673
C01753=1013.010,-110.084,-105.365,164.676,60.931,160.673
C01754=1013.015,-109.834,-105.372,164.679,60.927,160.672
C01755=1013.019,-109.584,-105.380,164.682,60.922,160.673
C01756=1013.023,-109.334,-105.387,164.684,60.917,160.672
C01757=1013.028,-109.084,-105.394,164.686,60.913,160.672
C01758=1013.032,-108.834,-105.402,164.689,60.908,160.672
C01759=1013.037,-108.584,-105.409,164.691,60.904,160.672
C01760=1013.042,-108.335,-105.416,164.694,60.898,160.672
C01761=1013.046,-108.086,-105.423,164.696,60.894,160.672
C01762=1013.051,-107.835,-105.431,164.697,60.889,160.671
C01763=1013.056,-107.586,-105.438,164.701,60.884,160.672
C01764=1013.060,-107.336,-105.446,164.702,60.880,160.671
C01765=1013.065,-107.086,-105.454,164.705,60.875,160.671
C01766=1013.069,-106.836,-105.462,164.707,60.870,160.671
C01767=1013.073,-106.586,-105.469,164.710,60.866,160.671
C01768=1013.077,-106.336,-105.476,164.712,60.860,160.671
C01769=1013.082,-106.086,-105.484,164.715,60.856,160.671
C01770=1013.087,-105.836,-105.492,164.717,60.851,160.670
C01771=1013.091,-105.587,-105.499,164.720,60.847,160.670
C01772=1013.096,-105.336,-105.507,164.721,60.842,160.670
C01773=1013.100,-105.087,-105.514,164.725,60.837,160.670
C01774=1013.105,-104.837,-105.522,164.726,60.832,160.670
C01775=1013.109,-104.588,-105.529,164.729,60.827,160.670
C01776=1013.114,-104.337,-105.537,164.731,60.823,160.670
C01777=1013.118,-104.088,-105.544,164.734,60.817,160.669
C01778=1013.123,-103.838,-105.552,164.735,60.813,160.669
C01779=1013.128,-103.588,-105.559,164.739,60.808,160.669
C01780=1013.131,-103.338,-105.567,164.740,60.803,160.669
C01781=1013.136,-103.089,-105.575,164.743,60.798,160.669
